C09136=1200.928,251.672,-63.247,-177.101,6.857,148.420
C09137=1200.933,251.424,-63.219,-177.103,6.855,148.421
C09138=1200.938,251.175,-63.192,-177.105,6.853,148.421
C09139=1200.942,250.926,-63.167,-177.109,6.850,148.421
C09140=1200.947,250.678,-63.140,-177.111,6.848,148.421
C09141=1200.951,250.429,-63.112,-177.113,6.846,148.421
C09142=1200.955,250.180,-63.086,-177.116,6.843,148.421
C09143=1200.959,249.932,-63.059,-177.119,6.841,148.422
C09144=1200.964,249.683,-63.033,-177.121,6.839,148.422
C09145=1200.968,249.435,-63.006,-177.124,6.836,148.422
C09146=1200.973,249.186,-62.979,-177.126,6.834,148.422
C09147=1200.977,248.938,-62.952,-177.129,6.832,148.422
C09148=1200.982,248.689,-62.926,-177.131,6.830,148.423
C09149=1200.986,248.441,-62.900,-177.134,6.828,148.423
C09150=1200.990,248.192,-62.872,-177.136,6.825,148.423
C09151=1200.995,247.943,-62.846,-177.139,6.824,148.423
C09152=1200.999,247.695,-62.820,-177.142,6.821,148.423
C09153=1201.004,247.446,-62.793,-177.144,6.819,148.424
C09154=1201.009,247.198,-62.767,-177.147,6.817,148.424
C09155=1201.013,246.950,-62.740,-177.150,6.814,148.424
C09156=1201.017,246.702,-62.714,-177.152,6.812,148.424
C09157=1201.022,246.452,-62.687,-177.154,6.810,148.424
C09158=1201.026,246.204,-62.661,-177.157,6.808,148.424
C09159=1201.031,245.955,-62.635,-177.160,6.805,148.425
C09160=1201.035,245.707,-62.608,-177.162,6.803,148.425
C09161=1201.040,245.458,-62.581,-177.165,6.801,148.425
C09162=1201.044,245.210,-62.555,-177.168,6.798,148.425
C09163=1201.049,244.961,-62.528,-177.170,6.796,148.426
C09164=1201.053,244.712,-62.502,-177.173,6.794,148.426
C09165=1201.057,244.464,-62.475,-177.175,6.792,148.426
C09166=1201.062,244.215,-62.450,-177.178,6.789,148.426
C09167=1201.066,243.967,-62.423,-177.180,6.787,148.426
C09168=1201.071,243.718,-62.397,-177.183,6.785,148.427
C09169=1201.075,243.470,-62.371,-177.186,6.783,148.427
C09170=1201.080,243.221,-62.344,-177.188,6.781,148.427
C09171=1201.084,242.973,-62.318,-177.191,6.779,148.427
C09172=1201.089,242.724,-62.292,-177.193,6.777,148.427
C09173=1201.093,242.475,-62.266,-177.196,6.774,148.428
C09174=1201.097,242.227,-62.239,-177.198,6.772,148.428
C09175=1201.102,241.978,-62.213,-177.201,6.770,148.428
C09176=1201.106,241.730,-62.187,-177.203,6.768,148.428
C09177=1201.111,241.480,-62.160,-177.206,6.765,148.428
C09178=1201.116,241.232,-62.135,-177.209,6.763,148.429
C09179=1201.120,240.984,-62.108,-177.211,6.761,148.429
C09180=1201.125,240.735,-62.082,-177.214,6.759,148.429
C09181=1201.129,240.486,-62.056,-177.217,6.757,148.429
C09182=1201.133,240.238,-62.030,-177.219,6.754,148.430
C09183=1201.138,239.989,-62.003,-177.222,6.752,148.430
C09184=1201.143,239.741,-61.978,-177.224,6.750,148.430
C09185=1201.146,239.493,-61.952,-177.227,6.748,148.430
C09186=1201.151,239.243,-61.925,-177.230,6.746,148.431
C09187=1201.156,238.995,-61.899,-177.232,6.744,148.431
C09188=1201.160,238.746,-61.874,-177.234,6.742,148.431
C09189=1201.164,238.498,-61.848,-177.237,6.739,148.431
C09190=1201.169,238.249,-61.821,-177.240,6.737,148.431
C09191=1201.174,238.000,-61.796,-177.242,6.735,148.432
C09192=1201.178,237.752,-61.770,-177.244,6.733,148.432
C09193=1201.182,237.503,-61.743,-177.248,6.730,148.432
C09194=1201.188,237.232,-61.715,-177.250,6.728,148.432
C09195=1201.192,236.960,-61.687,-177.253,6.725,148.432
C09196=1201.197,236.689,-61.658,-177.256,6.724,148.433
C09197=1201.202,236.418,-61.631,-177.259,6.721,148.433
C09198=1201.206,236.169,-61.605,-177.262,6.719,148.433
C09199=1201.211,235.920,-61.578,-177.264,6.717,148.434
C09200=1201.215,235.671,-61.552,-177.266,6.715,148.434
C09201=1201.220,235.423,-61.527,-177.269,6.712,148.434
C09202=1201.224,235.175,-61.501,-177.272,6.710,148.434
C09203=1201.228,234.926,-61.475,-177.274,6.708,148.435
C09204=1201.233,234.677,-61.449,-177.276,6.706,148.435
C09205=1201.238,234.429,-61.423,-177.280,6.704,148.435
C09206=1201.242,234.180,-61.398,-177.282,6.702,148.435
C09207=1201.247,233.931,-61.372,-177.284,6.700,148.435
C09208=1201.252,233.683,-61.346,-177.287,6.698,148.436
C09209=1201.256,233.434,-61.321,-177.290,6.696,148.436
C09210=1201.260,233.185,-61.295,-177.292,6.693,148.436
C09211=1201.264,232.936,-61.269,-177.295,6.691,148.436
C09212=1201.269,232.688,-61.244,-177.298,6.689,148.437
C09213=1201.273,232.440,-61.218,-177.300,6.687,148.437
C09214=1201.278,232.190,-61.192,-177.302,6.685,148.437
C09215=1201.283,231.942,-61.166,-177.306,6.683,148.437
C09216=1201.287,231.694,-61.141,-177.308,6.680,148.438
C09217=1201.292,231.445,-61.115,-177.310,6.679,148.438
C09218=1201.296,231.197,-61.089,-177.313,6.677,148.438
C09219=1201.301,230.947,-61.064,-177.315,6.675,148.438
C09220=1201.305,230.698,-61.039,-177.318,6.672,148.439
C09221=1201.310,230.450,-61.013,-177.321,6.670,148.439
C09222=1201.314,230.201,-60.988,-177.323,6.668,148.439
C09223=1201.318,229.953,-60.962,-177.326,6.666,148.439
C09224=1201.323,229.705,-60.936,-177.329,6.664,148.440
C09225=1201.327,229.456,-60.911,-177.331,6.662,148.440
C09226=1201.333,229.207,-60.886,-177.334,6.659,148.440
C09227=1201.337,228.958,-60.860,-177.337,6.658,148.440
C09228=1201.341,228.709,-60.834,-177.339,6.656,148.441
C09229=1201.346,228.461,-60.809,-177.341,6.654,148.441
C09230=1201.350,228.212,-60.784,-177.344,6.652,148.441
C09231=1201.355,227.963,-60.758,-177.347,6.649,148.441
C09232=1201.359,227.715,-60.733,-177.349,6.647,148.442
C09233=1201.364,227.466,-60.707,-177.352,6.645,148.442
C09234=1201.369,227.217,-60.683,-177.355,6.643,148.442
C09235=1201.372,226.969,-60.657,-177.357,6.641,148.442
C09236=1201.376,226.720,-60.632,-177.359,6.639,148.443
C09237=1201.381,226.472,-60.606,-177.363,6.637,148.443
C09238=1201.386,226.223,-60.581,-177.365,6.635,148.443
C09239=1201.391,225.975,-60.556,-177.367,6.633,148.443
C09240=1201.395,225.726,-60.530,-177.370,6.631,148.444
C09241=1201.400,225.477,-60.505,-177.373,6.629,148.444
C09242=1201.404,225.228,-60.480,-177.375,6.627,148.444
C09243=1201.409,224.979,-60.455,-177.378,6.624,148.444
C09244=1201.413,224.731,-60.430,-177.381,6.622,148.445
C09245=1201.417,224.482,-60.404,-177.383,6.620,148.445
C09246=1201.422,224.233,-60.379,-177.386,6.619,148.445
C09247=1201.426,223.985,-60.354,-177.388,6.616,148.445
C09248=1201.432,223.736,-60.329,-177.391,6.615,148.446
C09249=1201.436,223.487,-60.303,-177.394,6.612,148.446
C09250=1201.440,223.239,-60.279,-177.396,6.610,148.446
C09251=1201.444,222.990,-60.253,-177.399,6.608,148.447
C09252=1201.450,222.741,-60.229,-177.401,6.606,148.447
C09253=1201.454,222.492,-60.203,-177.404,6.604,148.447
C09254=1201.459,222.244,-60.178,-177.407,6.602,148.448
C09255=1201.462,221.995,-60.153,-177.409,6.600,148.448
C09256=1201.468,221.746,-60.128,-177.412,6.598,148.448
C09257=1201.472,221.498,-60.103,-177.415,6.596,148.448
C09258=1201.477,221.249,-60.078,-177.417,6.594,148.449
C09259=1201.480,221.000,-60.053,-177.420,6.592,148.449
C09260=1201.485,220.752,-60.028,-177.422,6.590,148.449
C09261=1201.490,220.503,-60.002,-177.425,6.588,148.449
C09262=1201.494,220.254,-59.978,-177.427,6.586,148.450
C09263=1201.499,220.006,-59.954,-177.430,6.583,148.450
C09264=1201.503,219.757,-59.928,-177.433,6.581,148.450
C09265=1201.509,219.508,-59.903,-177.435,6.580,148.450
C09266=1201.512,219.259,-59.879,-177.438,6.578,148.451
C09267=1201.517,219.011,-59.853,-177.441,6.576,148.451
C09268=1201.522,218.762,-59.828,-177.443,6.574,148.451
C09269=1201.526,218.513,-59.804,-177.446,6.572,148.452
C09270=1201.530,218.264,-59.779,-177.448,6.570,148.452
C09271=1201.535,218.016,-59.754,-177.451,6.567,148.452
C09272=1201.540,217.767,-59.730,-177.454,6.565,148.452
C09273=1201.544,217.518,-59.704,-177.456,6.563,148.453
C09274=1201.549,217.270,-59.680,-177.459,6.562,148.453
C09275=1201.553,217.021,-59.655,-177.461,6.560,148.453
C09276=1201.558,216.772,-59.630,-177.464,6.558,148.454
C09277=1201.562,216.524,-59.606,-177.467,6.556,148.454
C09278=1201.567,216.275,-59.581,-177.469,6.554,148.454
C09279=1201.571,216.026,-59.556,-177.472,6.551,148.454
C09280=1201.576,215.777,-59.531,-177.475,6.550,148.455
C09281=1201.581,215.528,-59.507,-177.477,6.548,148.455
C09282=1201.585,215.280,-59.482,-177.480,6.546,148.455
C09283=1201.589,215.031,-59.457,-177.482,6.544,148.455
C09284=1201.594,214.782,-59.433,-177.485,6.542,148.456
C09285=1201.599,214.534,-59.408,-177.488,6.540,148.456
C09286=1201.603,214.285,-59.384,-177.490,6.538,148.456
C09287=1201.608,214.036,-59.359,-177.493,6.536,148.457
C09288=1201.612,213.787,-59.335,-177.496,6.534,148.457
C09289=1201.617,213.538,-59.310,-177.498,6.532,148.457
C09290=1201.621,213.290,-59.285,-177.501,6.530,148.458
C09291=1201.626,213.042,-59.261,-177.503,6.528,148.458
C09292=1201.630,212.792,-59.236,-177.506,6.526,148.458
C09293=1201.635,212.544,-59.211,-177.509,6.524,148.459
C09294=1201.639,212.295,-59.187,-177.511,6.522,148.459
C09295=1201.644,212.046,-59.162,-177.514,6.520,148.459
C09296=1201.648,211.797,-59.138,-177.516,6.518,148.459
C09297=1201.653,211.549,-59.114,-177.519,6.517,148.460
C09298=1201.658,211.278,-59.086,-177.522,6.514,148.460
C09299=1201.663,211.007,-59.061,-177.525,6.512,148.460
C09300=1201.668,210.737,-59.034,-177.527,6.510,148.461
C09301=1201.673,210.467,-59.008,-177.531,6.508,148.461
C09302=1201.678,210.218,-58.983,-177.533,6.506,148.461
C09303=1201.682,209.969,-58.959,-177.536,6.504,148.462
C09304=1201.686,209.721,-58.934,-177.539,6.502,148.462
C09305=1201.691,209.472,-58.910,-177.541,6.500,148.462
C09306=1201.695,209.223,-58.885,-177.543,6.498,148.462
C09307=1201.700,208.974,-58.862,-177.546,6.496,148.463
C09308=1201.705,208.725,-58.837,-177.549,6.495,148.463
C09309=1201.709,208.477,-58.813,-177.551,6.493,148.463
C09310=1201.715,208.228,-58.789,-177.554,6.491,148.464
C09311=1201.718,207.979,-58.764,-177.557,6.488,148.464
C09312=1201.723,207.731,-58.740,-177.560,6.486,148.464
C09313=1201.728,207.482,-58.715,-177.562,6.484,148.465
C09314=1201.733,207.233,-58.692,-177.565,6.482,148.465
C09315=1201.736,206.984,-58.668,-177.567,6.481,148.465
C09316=1201.742,206.735,-58.643,-177.570,6.479,148.466
C09317=1201.746,206.487,-58.619,-177.573,6.477,148.466
C09318=1201.751,206.237,-58.595,-177.575,6.475,148.466
C09319=1201.755,205.989,-58.571,-177.578,6.473,148.467
C09320=1201.760,205.740,-58.546,-177.581,6.472,148.467
C09321=1201.764,205.491,-58.522,-177.583,6.469,148.467
C09322=1201.769,205.242,-58.499,-177.585,6.468,148.467
C09323=1201.774,204.993,-58.474,-177.588,6.466,148.468
C09324=1201.778,204.745,-58.450,-177.591,6.464,148.468
C09325=1201.783,204.496,-58.427,-177.593,6.462,148.468
C09326=1201.787,204.247,-58.402,-177.596,6.460,148.469
C09327=1201.791,203.999,-58.378,-177.599,6.458,148.469
C09328=1201.797,203.749,-58.354,-177.601,6.457,148.469
C09329=1201.801,203.501,-58.330,-177.604,6.455,148.470
C09330=1201.805,203.252,-58.306,-177.606,6.453,148.470
C09331=1201.810,203.003,-58.283,-177.609,6.451,148.470
C09332=1201.814,202.755,-58.259,-177.611,6.449,148.471
C09333=1201.819,202.505,-58.234,-177.615,6.446,148.471
C09334=1201.824,202.256,-58.210,-177.617,6.445,148.471
C09335=1201.828,202.008,-58.186,-177.620,6.443,148.472
C09336=1201.833,201.759,-58.163,-177.623,6.441,148.472
C09337=1201.837,201.511,-58.139,-177.625,6.439,148.472
C09338=1201.842,201.262,-58.116,-177.628,6.437,148.473
C09339=1201.847,201.013,-58.091,-177.630,6.435,148.473
C09340=1201.852,200.764,-58.068,-177.633,6.434,148.473
C09341=1201.855,200.515,-58.043,-177.635,6.431,148.473
C09342=1201.860,200.266,-58.020,-177.638,6.430,148.474
C09343=1201.865,200.017,-57.996,-177.641,6.428,148.474
C09344=1201.869,199.768,-57.972,-177.643,6.426,148.474
C09345=1201.874,199.520,-57.948,-177.646,6.424,148.475
C09346=1201.878,199.271,-57.925,-177.649,6.422,148.475
C09347=1201.883,199.022,-57.901,-177.651,6.421,148.475
C09348=1201.887,198.773,-57.877,-177.654,6.419,148.476
C09349=1201.892,198.525,-57.853,-177.657,6.417,148.476
C09350=1201.897,198.276,-57.829,-177.659,6.415,148.477
C09351=1201.902,198.027,-57.806,-177.662,6.413,148.477
C09352=1201.906,197.778,-57.782,-177.664,6.411,148.477
C09353=1201.911,197.529,-57.759,-177.667,6.410,148.478
C09354=1201.915,197.281,-57.735,-177.670,6.408,148.478
C09355=1201.920,197.032,-57.711,-177.672,6.406,148.478
C09356=1201.925,196.783,-57.688,-177.675,6.404,148.478
C09357=1201.929,196.534,-57.664,-177.677,6.402,148.479
C09358=1201.934,196.285,-57.640,-177.680,6.400,148.479
C09359=1201.939,196.036,-57.617,-177.683,6.398,148.479
C09360=1201.943,195.787,-57.594,-177.685,6.397,148.480
C09361=1201.948,195.539,-57.570,-177.688,6.395,148.480
C09362=1201.952,195.290,-57.546,-177.691,6.393,148.480
C09363=1201.957,195.041,-57.523,-177.693,6.391,148.481
C09364=1201.962,194.792,-57.499,-177.696,6.389,148.481
C09365=1201.966,194.543,-57.475,-177.698,6.388,148.482
C09366=1201.970,194.294,-57.453,-177.701,6.387,148.482
C09367=1201.975,194.045,-57.429,-177.703,6.385,148.482
C09368=1201.980,193.796,-57.406,-177.706,6.383,148.483
C09369=1201.984,193.548,-57.382,-177.709,6.381,148.483
C09370=1201.989,193.299,-57.358,-177.711,6.379,148.483
C09371=1201.993,193.050,-57.335,-177.714,6.377,148.484
C09372=1201.998,192.801,-57.312,-177.717,6.376,148.484
C09373=1202.003,192.552,-57.288,-177.719,6.374,148.484
C09374=1202.007,192.303,-57.265,-177.722,6.372,148.485
C09375=1202.012,192.054,-57.241,-177.724,6.370,148.485
C09376=1202.016,191.806,-57.218,-177.727,6.368,148.485
C09377=1202.021,191.557,-57.195,-177.730,6.367,148.486
C09378=1202.025,191.308,-57.172,-177.732,6.365,148.486
C09379=1202.030,191.059,-57.148,-177.735,6.363,148.486
C09380=1202.035,190.810,-57.125,-177.738,6.361,148.487
C09381=1202.040,190.561,-57.102,-177.740,6.359,148.487
C09382=1202.045,190.312,-57.078,-177.743,6.357,148.487
C09383=1202.049,190.063,-57.056,-177.746,6.356,148.488
C09384=1202.053,189.814,-57.032,-177.748,6.354,148.488
C09385=1202.058,189.565,-57.009,-177.751,6.352,148.489
C09386=1202.063,189.316,-56.986,-177.754,6.350,148.489
C09387=1202.067,189.067,-56.962,-177.756,6.349,148.489
C09388=1202.071,188.819,-56.939,-177.758,6.347,148.490
C09389=1202.077,188.570,-56.916,-177.761,6.346,148.490
C09390=1202.081,188.321,-56.893,-177.764,6.344,148.490
C09391=1202.086,188.072,-56.870,-177.766,6.342,148.491
C09392=1202.090,187.823,-56.847,-177.769,6.340,148.491
C09393=1202.095,187.574,-56.824,-177.772,6.338,148.491
C09394=1202.099,187.325,-56.800,-177.774,6.337,148.492
C09395=1202.104,187.076,-56.777,-177.777,6.335,148.492
C09396=1202.109,186.828,-56.755,-177.780,6.333,148.492
C09397=1202.113,186.579,-56.731,-177.782,6.331,148.493
C09398=1202.118,186.330,-56.708,-177.785,6.329,148.493
C09399=1202.122,186.082,-56.685,-177.788,6.328,148.493
C09400=1202.127,185.832,-56.662,-177.790,6.326,148.494
C09401=1202.132,185.583,-56.639,-177.792,6.325,148.494
C09402=1202.136,185.313,-56.615,-177.796,6.322,148.495
C09403=1202.142,185.044,-56.590,-177.798,6.320,148.495
C09404=1202.147,184.775,-56.564,-177.801,6.318,148.495
C09405=1202.151,184.505,-56.539,-177.804,6.317,148.496
C09406=1202.157,184.256,-56.517,-177.806,6.315,148.496
C09407=1202.161,184.007,-56.494,-177.809,6.313,148.496
C09408=1202.166,183.758,-56.471,-177.812,6.312,148.497
C09409=1202.170,183.509,-56.448,-177.815,6.310,148.497
C09410=1202.174,183.260,-56.426,-177.817,6.308,148.498
C09411=1202.180,183.012,-56.403,-177.820,6.307,148.498
C09412=1202.184,182.763,-56.379,-177.822,6.305,148.498
C09413=1202.188,182.514,-56.356,-177.825,6.303,148.499
C09414=1202.193,182.264,-56.334,-177.828,6.302,148.499
C09415=1202.198,182.016,-56.311,-177.830,6.300,148.499
C09416=1202.203,181.767,-56.288,-177.833,6.298,148.500
C09417=1202.207,181.518,-56.266,-177.836,6.296,148.500
C09418=1202.212,181.269,-56.243,-177.838,6.294,148.500
C09419=1202.216,181.021,-56.220,-177.841,6.292,148.501
C09420=1202.221,180.771,-56.198,-177.843,6.292,148.501
C09421=1202.226,180.522,-56.174,-177.846,6.290,148.502
C09422=1202.230,180.273,-56.151,-177.848,6.288,148.502
C09423=1202.236,180.024,-56.129,-177.851,6.286,148.502
C09424=1202.239,179.776,-56.106,-177.854,6.284,148.503
C09425=1202.244,179.526,-56.084,-177.856,6.282,148.503
C09426=1202.249,179.278,-56.061,-177.859,6.281,148.503
C09427=1202.254,179.029,-56.038,-177.862,6.279,148.504
C09428=1202.258,178.780,-56.016,-177.864,6.278,148.504
C09429=1202.263,178.531,-55.993,-177.867,6.276,148.505
C09430=1202.268,178.282,-55.971,-177.869,6.275,148.505
C09431=1202.272,178.033,-55.948,-177.872,6.273,148.505
C09432=1202.277,177.784,-55.926,-177.875,6.271,148.506
C09433=1202.281,177.536,-55.903,-177.877,6.269,148.506
C09434=1202.286,177.286,-55.881,-177.880,6.267,148.506
C09435=1202.290,177.037,-55.858,-177.882,6.266,148.507
C09436=1202.296,176.788,-55.835,-177.885,6.265,148.507
C09437=1202.300,176.540,-55.813,-177.888,6.263,148.508
C09438=1202.305,176.291,-55.791,-177.890,6.261,148.508
C09439=1202.309,176.042,-55.768,-177.893,6.259,148.508
C09440=1202.313,175.793,-55.746,-177.896,6.257,148.509
C09441=1202.319,175.544,-55.723,-177.898,6.256,148.509
C09442=1202.323,175.295,-55.701,-177.901,6.255,148.510
C09443=1202.327,175.046,-55.679,-177.903,6.253,148.510
C09444=1202.333,174.797,-55.656,-177.906,6.251,148.510
C09445=1202.337,174.548,-55.633,-177.909,6.250,148.511
C09446=1202.343,174.299,-55.611,-177.911,6.248,148.511
C09447=1202.346,174.050,-55.588,-177.914,6.246,148.511
C09448=1202.351,173.801,-55.566,-177.916,6.245,148.512
C09449=1202.356,173.552,-55.544,-177.919,6.243,148.512
C09450=1202.360,173.303,-55.521,-177.922,6.241,148.513
C09451=1202.365,173.055,-55.500,-177.924,6.240,148.513
C09452=1202.369,172.805,-55.478,-177.927,6.238,148.513
C09453=1202.374,172.556,-55.454,-177.930,6.236,148.514
C09454=1202.379,172.308,-55.433,-177.932,6.235,148.514
C09455=1202.383,172.058,-55.411,-177.935,6.233,148.515
C09456=1202.389,171.809,-55.388,-177.937,6.232,148.515
C09457=1202.393,171.561,-55.365,-177.940,6.230,148.515
C09458=1202.398,171.312,-55.344,-177.943,6.228,148.516
C09459=1202.402,171.063,-55.322,-177.945,6.227,148.516
C09460=1202.407,170.813,-55.299,-177.948,6.225,148.516
C09461=1202.412,170.564,-55.277,-177.951,6.224,148.517
C09462=1202.416,170.316,-55.255,-177.953,6.222,148.517
C09463=1202.421,170.067,-55.233,-177.956,6.220,148.518
C09464=1202.426,169.817,-55.210,-177.959,6.218,148.518
C09465=1202.431,169.569,-55.189,-177.961,6.217,148.518
C09466=1202.435,169.319,-55.167,-177.963,6.216,148.519
C09467=1202.440,169.071,-55.145,-177.966,6.214,148.519
C09468=1202.444,168.822,-55.122,-177.969,6.212,148.520
C09469=1202.449,168.573,-55.100,-177.972,6.211,148.520
C09470=1202.454,168.324,-55.078,-177.974,6.210,148.521
C09471=1202.458,168.075,-55.056,-177.977,6.208,148.521
C09472=1202.463,167.826,-55.034,-177.979,6.206,148.521
C09473=1202.468,167.577,-55.012,-177.982,6.204,148.522
C09474=1202.473,167.327,-54.990,-177.984,6.203,148.522
C09475=1202.477,167.079,-54.968,-177.987,6.201,148.522
C09476=1202.482,166.829,-54.946,-177.990,6.200,148.523
C09477=1202.487,166.581,-54.924,-177.993,6.198,148.523
C09478=1202.491,166.331,-54.902,-177.995,6.196,148.524
C09479=1202.496,166.083,-54.881,-177.997,6.195,148.524
C09480=1202.500,165.833,-54.859,-178.000,6.194,148.524
C09481=1202.505,165.585,-54.837,-178.003,6.192,148.525
C09482=1202.510,165.336,-54.815,-178.005,6.190,148.525
C09483=1202.515,165.086,-54.793,-178.009,6.189,148.526
C09484=1202.520,164.838,-54.771,-178.011,6.188,148.526
C09485=1202.524,164.588,-54.749,-178.013,6.186,148.527
C09486=1202.529,164.340,-54.727,-178.016,6.184,148.527
C09487=1202.533,164.091,-54.705,-178.019,6.182,148.527
C09488=1202.538,163.842,-54.683,-178.021,6.181,148.528
C09489=1202.542,163.593,-54.661,-178.024,6.180,148.528
C09490=1202.547,163.344,-54.640,-178.027,6.178,148.529
C09491=1202.552,163.095,-54.618,-178.029,6.176,148.529
C09492=1202.556,162.846,-54.596,-178.031,6.175,148.529
C09493=1202.561,162.597,-54.575,-178.034,6.173,148.530
C09494=1202.566,162.347,-54.553,-178.037,6.172,148.530
C09495=1202.570,162.099,-54.531,-178.040,6.170,148.531
C09496=1202.575,161.850,-54.510,-178.042,6.169,148.531
C09497=1202.580,161.601,-54.488,-178.045,6.167,148.531
C09498=1202.584,161.352,-54.466,-178.047,6.166,148.532
C09499=1202.589,161.102,-54.445,-178.050,6.164,148.532
C09500=1202.594,160.853,-54.423,-178.052,6.163,148.533
C09501=1202.599,160.605,-54.401,-178.055,6.161,148.533
C09502=1202.603,160.355,-54.379,-178.058,6.160,148.534
C09503=1202.608,160.107,-54.357,-178.061,6.158,148.534
C09504=1202.613,159.858,-54.336,-178.063,6.157,148.534
C09505=1202.617,159.608,-54.314,-178.065,6.155,148.535
C09506=1202.622,159.339,-54.292,-178.069,6.154,148.535
C09507=1202.627,159.070,-54.268,-178.071,6.152,148.536
C09508=1202.632,158.801,-54.245,-178.074,6.150,148.536
C09509=1202.637,158.532,-54.221,-178.077,6.149,148.537
C09510=1202.642,158.283,-54.200,-178.080,6.147,148.537
C09511=1202.647,158.035,-54.178,-178.082,6.146,148.537
C09512=1202.652,157.785,-54.157,-178.085,6.144,148.538
C09513=1202.656,157.536,-54.136,-178.088,6.143,148.538
C09514=1202.661,157.288,-54.114,-178.090,6.141,148.539
C09515=1202.666,157.039,-54.093,-178.092,6.140,148.539
C09516=1202.670,156.789,-54.071,-178.095,6.138,148.540
C09517=1202.675,156.540,-54.050,-178.098,6.137,148.540
C09518=1202.680,156.291,-54.028,-178.101,6.135,148.540
C09519=1202.685,156.042,-54.006,-178.103,6.134,148.541
C09520=1202.689,155.793,-53.986,-178.106,6.132,148.541
C09521=1202.694,155.544,-53.964,-178.108,6.130,148.542
C09522=1202.699,155.295,-53.943,-178.111,6.130,148.542
C09523=1202.703,155.046,-53.921,-178.114,6.128,148.543
C09524=1202.708,154.797,-53.900,-178.116,6.126,148.543
C09525=1202.713,154.548,-53.879,-178.119,6.124,148.543
C09526=1202.717,154.300,-53.857,-178.121,6.123,148.544
C09527=1202.722,154.050,-53.836,-178.124,6.122,148.544
C09528=1202.727,153.801,-53.814,-178.127,6.120,148.545
C09529=1202.732,153.552,-53.793,-178.129,6.119,148.545
C09530=1202.736,153.303,-53.772,-178.132,6.117,148.546
C09531=1202.741,153.053,-53.751,-178.135,6.116,148.546
C09532=1202.746,152.804,-53.730,-178.137,6.115,148.547
C09533=1202.751,152.555,-53.708,-178.140,6.113,148.547
C09534=1202.755,152.307,-53.688,-178.142,6.111,148.547
C09535=1202.760,152.058,-53.666,-178.146,6.110,148.548
C09536=1202.765,151.808,-53.645,-178.148,6.109,148.548
C09537=1202.769,151.560,-53.624,-178.150,6.107,148.549
C09538=1202.774,151.310,-53.603,-178.153,6.105,148.549
C09539=1202.779,151.061,-53.582,-178.156,6.105,148.550
C09540=1202.784,150.812,-53.560,-178.158,6.103,148.550
C09541=1202.788,150.563,-53.540,-178.161,6.101,148.550
C09542=1202.793,150.314,-53.518,-178.163,6.100,148.551
C09543=1202.798,150.065,-53.497,-178.166,6.099,148.551
C09544=1202.802,149.816,-53.477,-178.169,6.097,148.552
C09545=1202.807,149.567,-53.455,-178.171,6.096,148.552
C09546=1202.812,149.317,-53.434,-178.174,6.094,148.553
C09547=1202.816,149.068,-53.413,-178.177,6.093,148.553
C09548=1202.821,148.819,-53.392,-178.179,6.092,148.554
C09549=1202.826,148.571,-53.371,-178.182,6.090,148.554
C09550=1202.831,148.322,-53.350,-178.184,6.088,148.554
C09551=1202.836,148.072,-53.329,-178.187,6.088,148.555
C09552=1202.840,147.824,-53.308,-178.190,6.086,148.555
C09553=1202.845,147.574,-53.287,-178.192,6.084,148.556
C09554=1202.849,147.325,-53.266,-178.194,6.083,148.556
C09555=1202.854,147.076,-53.245,-178.198,6.082,148.557
C09556=1202.859,146.827,-53.224,-178.200,6.080,148.557
C09557=1202.864,146.578,-53.203,-178.202,6.079,148.557
C09558=1202.869,146.329,-53.182,-178.205,6.077,148.558
C09559=1202.873,146.080,-53.162,-178.208,6.076,148.558
C09560=1202.878,145.831,-53.141,-178.210,6.075,148.559
C09561=1202.883,145.582,-53.121,-178.213,6.073,148.559
C09562=1202.887,145.332,-53.099,-178.216,6.071,148.560
C09563=1202.891,145.084,-53.078,-178.218,6.070,148.560
C09564=1202.897,144.834,-53.057,-178.221,6.069,148.561
C09565=1202.901,144.585,-53.037,-178.223,6.068,148.561
C09566=1202.906,144.336,-53.016,-178.226,6.066,148.562
C09567=1202.911,144.087,-52.996,-178.229,6.064,148.562
C09568=1202.916,143.838,-52.975,-178.231,6.063,148.562
C09569=1202.920,143.589,-52.954,-178.234,6.062,148.563
C09570=1202.925,143.340,-52.933,-178.237,6.060,148.563
C09571=1202.930,143.091,-52.913,-178.239,6.059,148.564
C09572=1202.935,142.842,-52.891,-178.242,6.058,148.564
C09573=1202.939,142.593,-52.871,-178.245,6.056,148.565
C09574=1202.944,142.344,-52.850,-178.247,6.055,148.565
C09575=1202.949,142.095,-52.830,-178.250,6.053,148.566
C09576=1202.953,141.845,-52.808,-178.252,6.053,148.566
C09577=1202.958,141.596,-52.788,-178.255,6.051,148.567
C09578=1202.962,141.347,-52.767,-178.258,6.049,148.567
C09579=1202.967,141.098,-52.746,-178.260,6.049,148.568
C09580=1202.972,140.849,-52.726,-178.263,6.047,148.568
C09581=1202.977,140.600,-52.705,-178.266,6.045,148.568
C09582=1202.982,140.351,-52.685,-178.268,6.044,148.569
C09583=1202.986,140.101,-52.665,-178.271,6.043,148.569
C09584=1202.991,139.852,-52.644,-178.273,6.042,148.570
C09585=1202.996,139.603,-52.624,-178.276,6.040,148.570
C09586=1203.001,139.354,-52.603,-178.279,6.038,148.571
C09587=1203.005,139.105,-52.582,-178.281,6.037,148.571
C09588=1203.010,138.856,-52.562,-178.284,6.036,148.571
C09589=1203.015,138.606,-52.541,-178.286,6.035,148.572
C09590=1203.020,138.357,-52.521,-178.289,6.033,148.573
C09591=1203.024,138.109,-52.500,-178.292,6.032,148.573
C09592=1203.030,137.860,-52.480,-178.294,6.031,148.574
C09593=1203.034,137.610,-52.460,-178.297,6.029,148.574
C09594=1203.039,137.361,-52.440,-178.299,6.028,148.574
C09595=1203.044,137.112,-52.419,-178.302,6.027,148.575
C09596=1203.049,136.863,-52.398,-178.305,6.025,148.575
C09597=1203.053,136.614,-52.378,-178.307,6.024,148.576
C09598=1203.058,136.364,-52.358,-178.310,6.023,148.576
C09599=1203.063,136.115,-52.337,-178.312,6.022,148.577
C09600=1203.067,135.866,-52.317,-178.315,6.020,148.577
C09601=1203.072,135.618,-52.297,-178.318,6.018,148.578
C09602=1203.077,135.368,-52.276,-178.320,6.017,148.578
C09603=1203.082,135.119,-52.256,-178.323,6.016,148.578
C09604=1203.086,134.870,-52.236,-178.325,6.015,148.579
C09605=1203.091,134.621,-52.215,-178.328,6.013,148.580
C09606=1203.096,134.371,-52.195,-178.330,6.012,148.580
C09607=1203.101,134.123,-52.175,-178.333,6.011,148.581
C09608=1203.106,133.874,-52.155,-178.336,6.009,148.581
C09609=1203.110,133.624,-52.135,-178.338,6.008,148.581
C09610=1203.116,133.356,-52.113,-178.341,6.007,148.582
C09611=1203.121,133.087,-52.092,-178.344,6.005,148.582
C09612=1203.125,132.818,-52.069,-178.347,6.004,148.583
C09613=1203.131,132.549,-52.047,-178.350,6.003,148.584
C09614=1203.136,132.301,-52.027,-178.353,6.001,148.584
C09615=1203.141,132.051,-52.007,-178.355,6.000,148.584
C09616=1203.145,131.802,-51.987,-178.358,5.999,148.585
C09617=1203.150,131.553,-51.967,-178.360,5.998,148.585
C09618=1203.154,131.304,-51.947,-178.363,5.996,148.586
C09619=1203.159,131.055,-51.927,-178.366,5.995,148.586
C09620=1203.164,130.805,-51.906,-178.368,5.994,148.587
C09621=1203.169,130.557,-51.886,-178.371,5.992,148.587
C09622=1203.174,130.308,-51.866,-178.373,5.991,148.588
C09623=1203.178,130.058,-51.846,-178.376,5.989,148.588
C09624=1203.183,129.809,-51.826,-178.379,5.989,148.589
C09625=1203.188,129.560,-51.806,-178.381,5.987,148.589
C09626=1203.192,129.311,-51.786,-178.383,5.986,148.590
C09627=1203.197,129.062,-51.767,-178.387,5.985,148.590
C09628=1203.202,128.813,-51.746,-178.389,5.983,148.591
C09629=1203.207,128.563,-51.726,-178.391,5.982,148.591
C09630=1203.212,128.314,-51.706,-178.394,5.981,148.592
C09631=1203.217,128.065,-51.686,-178.397,5.980,148.592
C09632=1203.222,127.816,-51.667,-178.400,5.978,148.593
C09633=1203.226,127.567,-51.646,-178.402,5.977,148.593
C09634=1203.231,127.317,-51.627,-178.405,5.975,148.593
C09635=1203.235,127.068,-51.606,-178.407,5.975,148.594
C09636=1203.241,126.819,-51.587,-178.410,5.973,148.594
C09637=1203.245,126.570,-51.567,-178.412,5.973,148.595
C09638=1203.250,126.321,-51.547,-178.415,5.971,148.596
C09639=1203.255,126.071,-51.527,-178.417,5.970,148.596
C09640=1203.259,125.822,-51.507,-178.420,5.968,148.597
C09641=1203.265,125.574,-51.488,-178.423,5.967,148.597
C09642=1203.269,125.324,-51.468,-178.425,5.966,148.597
C09643=1203.274,125.075,-51.448,-178.428,5.965,148.598
C09644=1203.278,124.825,-51.428,-178.431,5.963,148.598
C09645=1203.284,124.577,-51.409,-178.434,5.962,148.599
C09646=1203.288,124.328,-51.388,-178.436,5.961,148.599
C09647=1203.293,124.078,-51.369,-178.439,5.959,148.600
C09648=1203.298,123.829,-51.349,-178.441,5.959,148.600
C09649=1203.303,123.580,-51.329,-178.444,5.957,148.601
C09650=1203.307,123.331,-51.310,-178.446,5.956,148.601
C09651=1203.312,123.081,-51.290,-178.449,5.954,148.602
C09652=1203.317,122.833,-51.271,-178.452,5.954,148.602
C09653=1203.321,122.584,-51.251,-178.454,5.952,148.603
C09654=1203.326,122.334,-51.231,-178.457,5.951,148.603
C09655=1203.331,122.085,-51.212,-178.460,5.950,148.604
C09656=1203.336,121.836,-51.192,-178.462,5.949,148.604
C09657=1203.341,121.587,-51.172,-178.465,5.947,148.605
C09658=1203.346,121.338,-51.152,-178.467,5.946,148.605
C09659=1203.351,121.088,-51.133,-178.470,5.945,148.606
C09660=1203.355,120.839,-51.114,-178.472,5.944,148.606
C09661=1203.360,120.590,-51.094,-178.475,5.942,148.607
C09662=1203.365,120.341,-51.075,-178.478,5.942,148.607
C09663=1203.369,120.092,-51.054,-178.480,5.940,148.608
C09664=1203.375,119.843,-51.035,-178.483,5.939,148.608
C09665=1203.379,119.593,-51.015,-178.486,5.937,148.609
C09666=1203.383,119.344,-50.996,-178.488,5.937,148.609
C09667=1203.389,119.095,-50.977,-178.491,5.936,148.610
C09668=1203.393,118.845,-50.957,-178.493,5.934,148.610
C09669=1203.398,118.596,-50.938,-178.496,5.934,148.611
C09670=1203.403,118.347,-50.918,-178.499,5.932,148.611
C09671=1203.408,118.097,-50.899,-178.501,5.931,148.612
C09672=1203.412,117.850,-50.879,-178.504,5.929,148.612
C09673=1203.417,117.600,-50.860,-178.506,5.929,148.613
C09674=1203.422,117.350,-50.840,-178.509,5.927,148.613
C09675=1203.427,117.101,-50.821,-178.511,5.926,148.614
C09676=1203.431,116.852,-50.802,-178.514,5.925,148.614
C09677=1203.437,116.603,-50.782,-178.517,5.924,148.615
C09678=1203.441,116.354,-50.763,-178.520,5.922,148.615
C09679=1203.446,116.104,-50.743,-178.522,5.921,148.616
C09680=1203.451,115.856,-50.724,-178.525,5.920,148.616
C09681=1203.455,115.606,-50.705,-178.527,5.919,148.617
C09682=1203.461,115.357,-50.685,-178.530,5.918,148.618
C09683=1203.466,115.108,-50.666,-178.532,5.917,148.618
C09684=1203.470,114.858,-50.647,-178.535,5.916,148.618
C09685=1203.475,114.609,-50.628,-178.538,5.914,148.619
C09686=1203.480,114.359,-50.609,-178.540,5.913,148.619
C09687=1203.485,114.111,-50.590,-178.543,5.912,148.620
C09688=1203.489,113.861,-50.570,-178.545,5.911,148.620
C09689=1203.495,113.612,-50.551,-178.548,5.910,148.621
C09690=1203.499,113.363,-50.532,-178.550,5.909,148.621
C09691=1203.504,113.114,-50.513,-178.554,5.907,148.622
C09692=1203.509,112.865,-50.493,-178.556,5.906,148.623
C09693=1203.513,112.616,-50.474,-178.558,5.906,148.623
C09694=1203.518,112.366,-50.455,-178.561,5.904,148.624
C09695=1203.524,112.117,-50.436,-178.564,5.903,148.624
C09696=1203.528,111.868,-50.417,-178.566,5.902,148.625
C09697=1203.533,111.619,-50.398,-178.569,5.901,148.625
C09698=1203.538,111.369,-50.378,-178.572,5.899,148.626
C09699=1203.542,111.119,-50.360,-178.574,5.898,148.626
C09700=1203.548,110.871,-50.340,-178.577,5.897,148.627
C09701=1203.552,110.621,-50.321,-178.579,5.896,148.627
C09702=1203.557,110.373,-50.302,-178.582,5.895,148.628
C09703=1203.562,110.124,-50.283,-178.584,5.894,148.628
C09704=1203.567,109.874,-50.264,-178.587,5.893,148.629
C09705=1203.572,109.625,-50.245,-178.590,5.891,148.629
C09706=1203.576,109.376,-50.226,-178.592,5.891,148.630
C09707=1203.582,109.126,-50.207,-178.595,5.890,148.630
C09708=1203.586,108.877,-50.188,-178.598,5.888,148.631
C09709=1203.591,108.628,-50.169,-178.600,5.887,148.631
C09710=1203.595,108.379,-50.150,-178.603,5.886,148.632
C09711=1203.601,108.129,-50.131,-178.605,5.885,148.632
C09712=1203.605,107.880,-50.112,-178.608,5.884,148.633
C09713=1203.610,107.631,-50.093,-178.610,5.883,148.633
C09714=1203.615,107.362,-50.073,-178.614,5.881,148.634
C09715=1203.620,107.094,-50.053,-178.616,5.881,148.635
C09716=1203.626,106.826,-50.033,-178.619,5.879,148.635
C09717=1203.631,106.557,-50.011,-178.622,5.878,148.636
C09718=1203.636,106.308,-49.993,-178.625,5.877,148.636
C09719=1203.640,106.058,-49.974,-178.627,5.876,148.637
C09720=1203.645,105.810,-49.955,-178.630,5.875,148.637
C09721=1203.651,105.560,-49.937,-178.632,5.874,148.638
C09722=1203.655,105.311,-49.917,-178.635,5.873,148.638
C09723=1203.659,105.062,-49.900,-178.638,5.871,148.639
C09724=1203.664,104.812,-49.880,-178.640,5.871,148.639
C09725=1203.669,104.563,-49.862,-178.643,5.869,148.640
C09726=1203.674,104.314,-49.843,-178.645,5.868,148.641
C09727=1203.679,104.064,-49.824,-178.648,5.867,148.641
C09728=1203.684,103.815,-49.805,-178.651,5.866,148.642
C09729=1203.688,103.566,-49.787,-178.653,5.865,148.642
C09730=1203.693,103.317,-49.768,-178.656,5.865,148.643
C09731=1203.699,103.068,-49.749,-178.658,5.863,148.643
C09732=1203.703,102.818,-49.730,-178.661,5.862,148.644
C09733=1203.708,102.569,-49.712,-178.664,5.860,148.644
C09734=1203.713,102.320,-49.693,-178.666,5.860,148.645
C09735=1203.717,102.070,-49.675,-178.668,5.859,148.645
C09736=1203.723,101.822,-49.655,-178.671,5.858,148.646
C09737=1203.727,101.572,-49.637,-178.674,5.857,148.646
C09738=1203.731,101.323,-49.618,-178.676,5.856,148.647
C09739=1203.737,101.074,-49.600,-178.679,5.854,148.647
C09740=1203.742,100.824,-49.582,-178.682,5.854,148.648
C09741=1203.746,100.575,-49.563,-178.684,5.852,148.648
C09742=1203.752,100.326,-49.544,-178.687,5.851,148.649
C09743=1203.756,100.077,-49.525,-178.689,5.850,148.649
C09744=1203.761,99.827,-49.507,-178.692,5.849,148.650
C09745=1203.766,99.578,-49.489,-178.695,5.848,148.651
C09746=1203.771,99.329,-49.470,-178.697,5.847,148.651
C09747=1203.775,99.079,-49.451,-178.700,5.846,148.652
C09748=1203.781,98.830,-49.433,-178.702,5.845,148.652
C09749=1203.785,98.581,-49.414,-178.705,5.844,148.653
C09750=1203.790,98.331,-49.396,-178.708,5.843,148.653
C09751=1203.795,98.082,-49.378,-178.710,5.842,148.654
C09752=1203.800,97.833,-49.359,-178.713,5.840,148.654
C09753=1203.805,97.584,-49.341,-178.715,5.840,148.655
C09754=1203.809,97.334,-49.322,-178.718,5.839,148.655
C09755=1203.814,97.085,-49.304,-178.721,5.838,148.656
C09756=1203.819,96.836,-49.285,-178.723,5.837,148.656
C09757=1203.824,96.587,-49.267,-178.726,5.836,148.657
C09758=1203.829,96.337,-49.249,-178.729,5.835,148.658
C09759=1203.834,96.088,-49.231,-178.731,5.834,148.658
C09760=1203.838,95.839,-49.212,-178.733,5.833,148.659
C09761=1203.844,95.590,-49.193,-178.736,5.831,148.659
C09762=1203.848,95.340,-49.175,-178.739,5.831,148.660
C09763=1203.853,95.091,-49.157,-178.741,5.830,148.660
C09764=1203.858,94.842,-49.139,-178.744,5.829,148.661
C09765=1203.863,94.593,-49.120,-178.746,5.828,148.661
C09766=1203.868,94.343,-49.101,-178.749,5.827,148.662
C09767=1203.873,94.094,-49.083,-178.752,5.826,148.663
C09768=1203.877,93.845,-49.066,-178.754,5.825,148.663
C09769=1203.882,93.595,-49.048,-178.757,5.824,148.664
C09770=1203.887,93.346,-49.030,-178.760,5.822,148.664
C09771=1203.892,93.096,-49.011,-178.762,5.822,148.665
C09772=1203.897,92.847,-48.993,-178.764,5.821,148.665
C09773=1203.902,92.598,-48.974,-178.767,5.819,148.666
C09774=1203.907,92.349,-48.956,-178.770,5.819,148.666
C09775=1203.912,92.100,-48.938,-178.772,5.818,148.667
C09776=1203.916,91.850,-48.920,-178.775,5.817,148.667
C09777=1203.921,91.601,-48.902,-178.778,5.816,148.668
C09778=1203.926,91.352,-48.884,-178.780,5.815,148.669
C09779=1203.931,91.103,-48.866,-178.783,5.813,148.669
C09780=1203.936,90.853,-48.848,-178.786,5.813,148.670
C09781=1203.941,90.604,-48.830,-178.788,5.812,148.670
C09782=1203.945,90.354,-48.811,-178.790,5.811,148.671
C09783=1203.950,90.105,-48.793,-178.793,5.810,148.671
C09784=1203.955,89.856,-48.775,-178.796,5.809,148.672
C09785=1203.960,89.607,-48.757,-178.798,5.808,148.672
C09786=1203.965,89.357,-48.739,-178.801,5.807,148.673
C09787=1203.970,89.108,-48.721,-178.804,5.806,148.673
C09788=1203.975,88.859,-48.703,-178.806,5.805,148.674
C09789=1203.979,88.609,-48.685,-178.809,5.804,148.675
C09790=1203.984,88.360,-48.667,-178.812,5.803,148.675
C09791=1203.989,88.111,-48.649,-178.814,5.802,148.676
C09792=1203.994,87.862,-48.631,-178.816,5.802,148.676
C09793=1203.999,87.612,-48.613,-178.819,5.800,148.677
C09794=1204.004,87.363,-48.595,-178.822,5.799,148.677
C09795=1204.009,87.113,-48.577,-178.824,5.799,148.678
C09796=1204.014,86.864,-48.559,-178.827,5.797,148.678
C09797=1204.019,86.615,-48.541,-178.830,5.796,148.679
C09798=1204.023,86.365,-48.523,-178.832,5.796,148.680
C09799=1204.028,86.116,-48.505,-178.834,5.795,148.680
C09800=1204.032,85.867,-48.488,-178.838,5.794,148.681
C09801=1204.037,85.618,-48.470,-178.840,5.793,148.681
C09802=1204.043,85.368,-48.452,-178.842,5.792,148.682
C09803=1204.047,85.119,-48.435,-178.845,5.791,148.683
C09804=1204.052,84.870,-48.417,-178.848,5.790,148.683
C09805=1204.057,84.621,-48.399,-178.850,5.789,148.684
C09806=1204.062,84.372,-48.381,-178.852,5.788,148.684
C09807=1204.067,84.122,-48.363,-178.856,5.787,148.685
C09808=1204.072,83.873,-48.345,-178.858,5.786,148.685
C09809=1204.077,83.623,-48.327,-178.860,5.785,148.686
C09810=1204.082,83.374,-48.309,-178.864,5.784,148.686
C09811=1204.087,83.124,-48.292,-178.866,5.783,148.687
C09812=1204.092,82.876,-48.275,-178.868,5.782,148.687
C09813=1204.096,82.626,-48.257,-178.871,5.782,148.688
C09814=1204.101,82.377,-48.239,-178.874,5.780,148.689
C09815=1204.107,82.127,-48.222,-178.876,5.780,148.689
C09816=1204.111,81.878,-48.204,-178.879,5.779,148.690
C09817=1204.116,81.629,-48.186,-178.881,5.778,148.690
C09818=1204.122,81.360,-48.167,-178.884,5.777,148.691
C09819=1204.127,81.092,-48.147,-178.887,5.776,148.692
C09820=1204.132,80.823,-48.129,-178.890,5.775,148.692
C09821=1204.137,80.555,-48.110,-178.893,5.774,148.693
C09822=1204.142,80.306,-48.092,-178.895,5.773,148.693
C09823=1204.147,80.056,-48.075,-178.898,5.772,148.694
C09824=1204.152,79.807,-48.057,-178.900,5.771,148.694
C09825=1204.157,79.557,-48.039,-178.903,5.770,148.695
C09826=1204.161,79.308,-48.022,-178.905,5.770,148.696
C09827=1204.166,79.059,-48.004,-178.908,5.768,148.696
C09828=1204.171,78.809,-47.987,-178.911,5.768,148.697
C09829=1204.176,78.560,-47.969,-178.913,5.767,148.697
C09830=1204.181,78.311,-47.952,-178.915,5.766,148.698
C09831=1204.186,78.062,-47.935,-178.919,5.765,148.698
C09832=1204.191,77.813,-47.917,-178.921,5.764,148.699
C09833=1204.196,77.563,-47.899,-178.923,5.763,148.700
C09834=1204.200,77.314,-47.882,-178.926,5.763,148.700
C09835=1204.206,77.065,-47.865,-178.928,5.762,148.701
C09836=1204.210,76.815,-47.847,-178.931,5.760,148.701
C09837=1204.216,76.566,-47.829,-178.934,5.760,148.702
C09838=1204.220,76.317,-47.812,-178.936,5.759,148.702
C09839=1204.225,76.067,-47.795,-178.939,5.758,148.703
C09840=1204.230,75.818,-47.777,-178.942,5.757,148.704
C09841=1204.234,75.568,-47.760,-178.944,5.756,148.704
C09842=1204.239,75.319,-47.742,-178.947,5.755,148.705
C09843=1204.245,75.069,-47.725,-178.949,5.755,148.705
C09844=1204.249,74.820,-47.708,-178.952,5.754,148.706
C09845=1204.255,74.571,-47.691,-178.955,5.753,148.707
C09846=1204.260,74.322,-47.673,-178.957,5.752,148.707
C09847=1204.264,74.073,-47.656,-178.960,5.751,148.708
C09848=1204.269,73.823,-47.639,-178.962,5.751,148.708
C09849=1204.274,73.573,-47.621,-178.965,5.749,148.709
C09850=1204.279,73.324,-47.604,-178.967,5.748,148.709
C09851=1204.284,73.074,-47.587,-178.970,5.748,148.710
C09852=1204.288,72.826,-47.569,-178.972,5.747,148.710
C09853=1204.294,72.577,-47.552,-178.975,5.746,148.711
C09854=1204.299,72.327,-47.535,-178.978,5.745,148.712
C09855=1204.303,72.078,-47.518,-178.980,5.744,148.712
C09856=1204.308,71.828,-47.501,-178.983,5.743,148.713
C09857=1204.313,71.579,-47.484,-178.985,5.743,148.714
C09858=1204.318,71.329,-47.466,-178.988,5.742,148.714
C09859=1204.323,71.080,-47.449,-178.991,5.741,148.715
C09860=1204.328,70.831,-47.432,-178.993,5.740,148.715
C09861=1204.333,70.582,-47.414,-178.996,5.739,148.716
C09862=1204.338,70.332,-47.398,-178.998,5.739,148.716
C09863=1204.343,70.082,-47.380,-179.001,5.738,148.717
C09864=1204.347,69.833,-47.364,-179.004,5.736,148.717
C09865=1204.352,69.584,-47.346,-179.006,5.736,148.718
C09866=1204.358,69.335,-47.329,-179.009,5.735,148.719
C09867=1204.362,69.085,-47.312,-179.011,5.734,148.719
C09868=1204.368,68.835,-47.295,-179.014,5.734,148.720
C09869=1204.372,68.586,-47.278,-179.017,5.732,148.721
C09870=1204.377,68.337,-47.260,-179.019,5.731,148.721
C09871=1204.382,68.088,-47.244,-179.022,5.731,148.722
C09872=1204.387,67.838,-47.227,-179.024,5.730,148.722
C09873=1204.392,67.589,-47.210,-179.026,5.729,148.723
C09874=1204.397,67.339,-47.192,-179.029,5.729,148.723
C09875=1204.401,67.090,-47.175,-179.032,5.727,148.724
C09876=1204.406,66.841,-47.159,-179.035,5.727,148.725
C09877=1204.412,66.591,-47.142,-179.037,5.726,148.725
C09878=1204.416,66.342,-47.125,-179.040,5.725,148.726
C09879=1204.421,66.092,-47.108,-179.042,5.725,148.726
C09880=1204.426,65.843,-47.092,-179.044,5.724,148.727
C09881=1204.431,65.594,-47.074,-179.048,5.723,148.728
C09882=1204.436,65.345,-47.057,-179.050,5.722,148.728
C09883=1204.441,65.095,-47.040,-179.052,5.721,148.729
C09884=1204.446,64.846,-47.023,-179.055,5.721,148.729
C09885=1204.450,64.597,-47.007,-179.058,5.720,148.730
C09886=1204.456,64.347,-46.989,-179.060,5.719,148.730
C09887=1204.460,64.097,-46.973,-179.063,5.718,148.731
C09888=1204.466,63.848,-46.956,-179.066,5.717,148.732
C09889=1204.470,63.599,-46.939,-179.068,5.716,148.732
C09890=1204.475,63.349,-46.923,-179.070,5.716,148.733
C09891=1204.481,63.100,-46.906,-179.073,5.715,148.733
C09892=1204.485,62.851,-46.889,-179.076,5.715,148.734
C09893=1204.490,62.601,-46.872,-179.078,5.713,148.735
C09894=1204.495,62.351,-46.855,-179.081,5.712,148.735
C09895=1204.500,62.103,-46.839,-179.084,5.712,148.736
C09896=1204.505,61.853,-46.821,-179.086,5.711,148.736
C09897=1204.510,61.603,-46.805,-179.088,5.710,148.737
C09898=1204.515,61.355,-46.789,-179.091,5.710,148.738
C09899=1204.520,61.105,-46.771,-179.093,5.709,148.738
C09900=1204.524,60.855,-46.755,-179.096,5.707,148.739
C09901=1204.530,60.606,-46.738,-179.099,5.707,148.739
C09902=1204.534,60.357,-46.722,-179.102,5.706,148.740
C09903=1204.539,60.107,-46.704,-179.104,5.705,148.741
C09904=1204.544,59.858,-46.688,-179.106,5.705,148.741
C09905=1204.549,59.609,-46.671,-179.109,5.704,148.742
C09906=1204.554,59.358,-46.655,-179.111,5.703,148.742
C09907=1204.559,59.110,-46.639,-179.114,5.702,148.743
C09908=1204.564,58.860,-46.622,-179.117,5.702,148.744
C09909=1204.568,58.611,-46.605,-179.120,5.701,148.744
C09910=1204.574,58.362,-46.588,-179.122,5.700,148.745
C09911=1204.579,58.112,-46.572,-179.124,5.700,148.745
C09912=1204.584,57.863,-46.555,-179.127,5.699,148.746
C09913=1204.589,57.613,-46.539,-179.129,5.698,148.746
C09914=1204.594,57.363,-46.522,-179.132,5.698,148.747
C09915=1204.599,57.115,-46.506,-179.135,5.696,148.748
C09916=1204.603,56.865,-46.489,-179.138,5.696,148.748
C09917=1204.608,56.616,-46.472,-179.140,5.695,148.749
C09918=1204.614,56.366,-46.456,-179.142,5.694,148.750
C09919=1204.618,56.117,-46.440,-179.145,5.694,148.750
C09920=1204.624,55.868,-46.423,-179.147,5.693,148.751
C09921=1204.628,55.618,-46.407,-179.150,5.692,148.751
C09922=1204.634,55.349,-46.389,-179.153,5.691,148.752
C09923=1204.639,55.081,-46.371,-179.156,5.690,148.753
C09924=1204.644,54.812,-46.354,-179.158,5.690,148.753
C09925=1204.650,54.545,-46.336,-179.161,5.689,148.754
C09926=1204.654,54.295,-46.319,-179.164,5.688,148.755
C09927=1204.660,54.045,-46.303,-179.166,5.687,148.755
C09928=1204.665,53.796,-46.287,-179.169,5.686,148.756
C09929=1204.669,53.546,-46.270,-179.172,5.686,148.756
C09930=1204.675,53.297,-46.254,-179.174,5.685,148.757
C09931=1204.679,53.048,-46.238,-179.176,5.684,148.758
C09932=1204.684,52.799,-46.221,-179.179,5.684,148.758
C09933=1204.689,52.549,-46.205,-179.182,5.683,148.759
C09934=1204.694,52.300,-46.189,-179.184,5.683,148.760
C09935=1204.699,52.050,-46.172,-179.186,5.682,148.760
C09936=1204.704,51.800,-46.156,-179.190,5.681,148.761
C09937=1204.709,51.551,-46.140,-179.192,5.680,148.761
C09938=1204.714,51.301,-46.124,-179.194,5.679,148.762
C09939=1204.719,51.052,-46.107,-179.197,5.679,148.762
C09940=1204.724,50.803,-46.091,-179.200,5.678,148.763
C09941=1204.729,50.553,-46.075,-179.202,5.677,148.764
C09942=1204.733,50.304,-46.058,-179.205,5.677,148.764
C09943=1204.739,50.055,-46.043,-179.207,5.676,148.765
C09944=1204.743,49.805,-46.026,-179.210,5.675,148.766
C09945=1204.749,49.556,-46.011,-179.212,5.675,148.766
C09946=1204.753,49.306,-45.994,-179.215,5.674,148.767
C09947=1204.758,49.057,-45.978,-179.217,5.673,148.767
C09948=1204.763,48.807,-45.962,-179.220,5.672,148.768
C09949=1204.768,48.558,-45.945,-179.223,5.672,148.769
C09950=1204.773,48.308,-45.929,-179.225,5.671,148.769
C09951=1204.778,48.060,-45.913,-179.228,5.670,148.770
C09952=1204.783,47.809,-45.897,-179.231,5.670,148.770
C09953=1204.788,47.561,-45.881,-179.233,5.669,148.771
C09954=1204.793,47.311,-45.865,-179.235,5.668,148.772
C09955=1204.798,47.061,-45.849,-179.238,5.668,148.772
C09956=1204.803,46.812,-45.833,-179.241,5.667,148.773
C09957=1204.808,46.562,-45.817,-179.243,5.667,148.774
C09958=1204.813,46.314,-45.801,-179.245,5.666,148.774
C09959=1204.818,46.063,-45.785,-179.248,5.665,148.775
C09960=1204.823,45.815,-45.769,-179.251,5.665,148.775
C09961=1204.828,45.565,-45.753,-179.253,5.664,148.776
C09962=1204.833,45.315,-45.737,-179.256,5.662,148.776
C09963=1204.838,45.066,-45.721,-179.259,5.662,148.777
C09964=1204.843,44.816,-45.705,-179.261,5.661,148.778
C09965=1204.848,44.567,-45.688,-179.264,5.661,148.778
C09966=1204.853,44.317,-45.672,-179.267,5.660,148.779
C09967=1204.858,44.068,-45.657,-179.269,5.659,148.780
C09968=1204.863,43.818,-45.640,-179.271,5.659,148.780
C09969=1204.868,43.569,-45.625,-179.274,5.658,148.781
C09970=1204.873,43.320,-45.610,-179.277,5.658,148.782
C09971=1204.877,43.071,-45.593,-179.279,5.657,148.782
C09972=1204.883,42.821,-45.577,-179.281,5.656,148.783
C09973=1204.888,42.572,-45.562,-179.284,5.656,148.783
C09974=1204.892,42.322,-45.545,-179.287,5.655,148.784
C09975=1204.898,42.073,-45.530,-179.289,5.654,148.785
C09976=1204.903,41.823,-45.514,-179.292,5.654,148.785
C09977=1204.908,41.573,-45.498,-179.294,5.653,148.786
C09978=1204.912,41.325,-45.482,-179.297,5.653,148.787
C09979=1204.917,41.075,-45.466,-179.299,5.652,148.787
C09980=1204.922,40.825,-45.451,-179.302,5.651,148.788
C09981=1204.928,40.576,-45.435,-179.304,5.651,148.788
C09982=1204.932,40.326,-45.418,-179.307,5.650,148.789
C09983=1204.938,40.077,-45.403,-179.310,5.649,148.790
C09984=1204.942,39.828,-45.388,-179.312,5.648,148.790
C09985=1204.947,39.578,-45.372,-179.315,5.647,148.791
C09986=1204.952,39.329,-45.356,-179.318,5.647,148.791
C09987=1204.958,39.080,-45.340,-179.320,5.646,148.792
C09988=1204.962,38.830,-45.324,-179.322,5.645,148.793
C09989=1204.967,38.580,-45.309,-179.325,5.645,148.793
C09990=1204.972,38.331,-45.294,-179.328,5.644,148.794
C09991=1204.977,38.081,-45.278,-179.330,5.644,148.795
C09992=1204.983,37.832,-45.262,-179.333,5.643,148.795
C09993=1204.987,37.583,-45.246,-179.335,5.642,148.796
C09994=1204.992,37.333,-45.230,-179.338,5.642,148.796
C09995=1204.997,37.084,-45.215,-179.340,5.641,148.797
C09996=1205.002,36.834,-45.199,-179.343,5.641,148.798
//INST
///DATE 2021/06/25 14:28
///ATTR SC,RW,RJ
////FRAME ROBOT
///GROUP1 RB1
NOP
MOVL C00000 V=800.0 PL=0
MOVL C00001 V=800.0 PL=0
MOVL C00002 V=800.0 PL=0
MOVL C00003 V=800.0 PL=0
MOVL C00004 V=800.0 PL=0
MOVL C00005 V=800.0 PL=0
MOVL C00006 V=800.0 PL=0
MOVL C00007 V=800.0 PL=0
MOVL C00008 V=800.0 PL=0
MOVL C00009 V=800.0 PL=0
MOVL C00010 V=800.0 PL=0
MOVL C00011 V=800.0 PL=0
MOVL C00012 V=800.0 PL=0
MOVL C00013 V=800.0 PL=0
MOVL C00014 V=800.0 PL=0
MOVL C00015 V=800.0 PL=0
MOVL C00016 V=800.0 PL=0
MOVL C00017 V=800.0 PL=0
MOVL C00018 V=800.0 PL=0
MOVL C00019 V=800.0 PL=0
MOVL C00020 V=800.0 PL=0
MOVL C00021 V=800.0 PL=0
MOVL C00022 V=800.0 PL=0
MOVL C00023 V=800.0 PL=0
MOVL C00024 V=800.0 PL=0
MOVL C00025 V=800.0 PL=0
MOVL C00026 V=800.0 PL=0
MOVL C00027 V=800.0 PL=0
MOVL C00028 V=800.0 PL=0
MOVL C00029 V=800.0 PL=0
MOVL C00030 V=800.0 PL=0
MOVL C00031 V=800.0 PL=0
MOVL C00032 V=800.0 PL=0
MOVL C00033 V=800.0 PL=0
MOVL C00034 V=800.0 PL=0
MOVL C00035 V=800.0 PL=0
MOVL C00036 V=800.0 PL=0
MOVL C00037 V=800.0 PL=0
MOVL C00038 V=800.0 PL=0
MOVL C00039 V=800.0 PL=0
MOVL C00040 V=800.0 PL=0
MOVL C00041 V=800.0 PL=0
MOVL C00042 V=800.0 PL=0
MOVL C00043 V=800.0 PL=0
MOVL C00044 V=800.0 PL=0
MOVL C00045 V=800.0 PL=0
MOVL C00046 V=800.0 PL=0
MOVL C00047 V=800.0 PL=0
MOVL C00048 V=800.0 PL=0
MOVL C00049 V=800.0 PL=0
MOVL C00050 V=800.0 PL=0
MOVL C00051 V=800.0 PL=0
MOVL C00052 V=800.0 PL=0
MOVL C00053 V=800.0 PL=0
MOVL C00054 V=800.0 PL=0
MOVL C00055 V=800.0 PL=0
MOVL C00056 V=800.0 PL=0
MOVL C00057 V=800.0 PL=0
MOVL C00058 V=800.0 PL=0
MOVL C00059 V=800.0 PL=0
MOVL C00060 V=800.0 PL=0
MOVL C00061 V=800.0 PL=0
MOVL C00062 V=800.0 PL=0
MOVL C00063 V=800.0 PL=0
MOVL C00064 V=800.0 PL=0
MOVL C00065 V=800.0 PL=0
MOVL C00066 V=800.0 PL=0
MOVL C00067 V=800.0 PL=0
MOVL C00068 V=800.0 PL=0
MOVL C00069 V=800.0 PL=0
MOVL C00070 V=800.0 PL=0
MOVL C00071 V=800.0 PL=0
MOVL C00072 V=800.0 PL=0
MOVL C00073 V=800.0 PL=0
MOVL C00074 V=800.0 PL=0
MOVL C00075 V=800.0 PL=0
MOVL C00076 V=800.0 PL=0
MOVL C00077 V=800.0 PL=0
MOVL C00078 V=800.0 PL=0
MOVL C00079 V=800.0 PL=0
MOVL C00080 V=800.0 PL=0
MOVL C00081 V=800.0 PL=0
MOVL C00082 V=800.0 PL=0
MOVL C00083 V=800.0 PL=0
MOVL C00084 V=800.0 PL=0
MOVL C00085 V=800.0 PL=0
MOVL C00086 V=800.0 PL=0
MOVL C00087 V=800.0 PL=0
MOVL C00088 V=800.0 PL=0
MOVL C00089 V=800.0 PL=0
MOVL C00090 V=800.0 PL=0
MOVL C00091 V=800.0 PL=0
MOVL C00092 V=800.0 PL=0
MOVL C00093 V=800.0 PL=0
MOVL C00094 V=800.0 PL=0
MOVL C00095 V=800.0 PL=0
MOVL C00096 V=800.0 PL=0
MOVL C00097 V=800.0 PL=0
MOVL C00098 V=800.0 PL=0
MOVL C00099 V=800.0 PL=0
MOVL C00100 V=800.0 PL=0
MOVL C00101 V=800.0 PL=0
MOVL C00102 V=800.0 PL=0
MOVL C00103 V=800.0 PL=0
MOVL C00104 V=800.0 PL=0
MOVL C00105 V=800.0 PL=0
MOVL C00106 V=800.0 PL=0
MOVL C00107 V=800.0 PL=0
MOVL C00108 V=800.0 PL=0
MOVL C00109 V=800.0 PL=0
MOVL C00110 V=800.0 PL=0
MOVL C00111 V=800.0 PL=0
MOVL C00112 V=800.0 PL=0
MOVL C00113 V=800.0 PL=0
MOVL C00114 V=800.0 PL=0
MOVL C00115 V=800.0 PL=0
MOVL C00116 V=800.0 PL=0
MOVL C00117 V=800.0 PL=0
MOVL C00118 V=800.0 PL=0
MOVL C00119 V=800.0 PL=0
MOVL C00120 V=800.0 PL=0
MOVL C00121 V=800.0 PL=0
MOVL C00122 V=800.0 PL=0
MOVL C00123 V=800.0 PL=0
MOVL C00124 V=800.0 PL=0
MOVL C00125 V=800.0 PL=0
MOVL C00126 V=800.0 PL=0
MOVL C00127 V=800.0 PL=0
MOVL C00128 V=800.0 PL=0
MOVL C00129 V=800.0 PL=0
MOVL C00130 V=800.0 PL=0
MOVL C00131 V=800.0 PL=0
MOVL C00132 V=800.0 PL=0
MOVL C00133 V=800.0 PL=0
MOVL C00134 V=800.0 PL=0
MOVL C00135 V=800.0 PL=0
MOVL C00136 V=800.0 PL=0
MOVL C00137 V=800.0 PL=0
MOVL C00138 V=800.0 PL=0
MOVL C00139 V=800.0 PL=0
MOVL C00140 V=800.0 PL=0
MOVL C00141 V=800.0 PL=0
MOVL C00142 V=800.0 PL=0
MOVL C00143 V=800.0 PL=0
MOVL C00144 V=800.0 PL=0
MOVL C00145 V=800.0 PL=0
MOVL C00146 V=800.0 PL=0
MOVL C00147 V=800.0 PL=0
MOVL C00148 V=800.0 PL=0
MOVL C00149 V=800.0 PL=0
MOVL C00150 V=800.0 PL=0
MOVL C00151 V=800.0 PL=0
MOVL C00152 V=800.0 PL=0
MOVL C00153 V=800.0 PL=0
MOVL C00154 V=800.0 PL=0
MOVL C00155 V=800.0 PL=0
MOVL C00156 V=800.0 PL=0
MOVL C00157 V=800.0 PL=0
MOVL C00158 V=800.0 PL=0
MOVL C00159 V=800.0 PL=0
MOVL C00160 V=800.0 PL=0
MOVL C00161 V=800.0 PL=0
MOVL C00162 V=800.0 PL=0
MOVL C00163 V=800.0 PL=0
MOVL C00164 V=800.0 PL=0
MOVL C00165 V=800.0 PL=0
MOVL C00166 V=800.0 PL=0
MOVL C00167 V=800.0 PL=0
MOVL C00168 V=800.0 PL=0
MOVL C00169 V=800.0 PL=0
MOVL C00170 V=800.0 PL=0
MOVL C00171 V=800.0 PL=0
MOVL C00172 V=800.0 PL=0
MOVL C00173 V=800.0 PL=0
MOVL C00174 V=800.0 PL=0
MOVL C00175 V=800.0 PL=0
MOVL C00176 V=800.0 PL=0
MOVL C00177 V=800.0 PL=0
MOVL C00178 V=800.0 PL=0
MOVL C00179 V=800.0 PL=0
MOVL C00180 V=800.0 PL=0
MOVL C00181 V=800.0 PL=0
MOVL C00182 V=800.0 PL=0
MOVL C00183 V=800.0 PL=0
MOVL C00184 V=800.0 PL=0
MOVL C00185 V=800.0 PL=0
MOVL C00186 V=800.0 PL=0
MOVL C00187 V=800.0 PL=0
MOVL C00188 V=800.0 PL=0
MOVL C00189 V=800.0 PL=0
MOVL C00190 V=800.0 PL=0
MOVL C00191 V=800.0 PL=0
MOVL C00192 V=800.0 PL=0
MOVL C00193 V=800.0 PL=0
MOVL C00194 V=800.0 PL=0
MOVL C00195 V=800.0 PL=0
MOVL C00196 V=800.0 PL=0
MOVL C00197 V=800.0 PL=0
MOVL C00198 V=800.0 PL=0
MOVL C00199 V=800.0 PL=0
MOVL C00200 V=800.0 PL=0
MOVL C00201 V=800.0 PL=0
MOVL C00202 V=800.0 PL=0
MOVL C00203 V=800.0 PL=0
MOVL C00204 V=800.0 PL=0
MOVL C00205 V=800.0 PL=0
MOVL C00206 V=800.0 PL=0
MOVL C00207 V=800.0 PL=0
MOVL C00208 V=800.0 PL=0
MOVL C00209 V=800.0 PL=0
MOVL C00210 V=800.0 PL=0
MOVL C00211 V=800.0 PL=0
MOVL C00212 V=800.0 PL=0
MOVL C00213 V=800.0 PL=0
MOVL C00214 V=800.0 PL=0
MOVL C00215 V=800.0 PL=0
MOVL C00216 V=800.0 PL=0
MOVL C00217 V=800.0 PL=0
MOVL C00218 V=800.0 PL=0
MOVL C00219 V=800.0 PL=0
MOVL C00220 V=800.0 PL=0
MOVL C00221 V=800.0 PL=0
MOVL C00222 V=800.0 PL=0
MOVL C00223 V=800.0 PL=0
MOVL C00224 V=800.0 PL=0
MOVL C00225 V=800.0 PL=0
MOVL C00226 V=800.0 PL=0
MOVL C00227 V=800.0 PL=0
MOVL C00228 V=800.0 PL=0
MOVL C00229 V=800.0 PL=0
MOVL C00230 V=800.0 PL=0
MOVL C00231 V=800.0 PL=0
MOVL C00232 V=800.0 PL=0
MOVL C00233 V=800.0 PL=0
MOVL C00234 V=800.0 PL=0
MOVL C00235 V=800.0 PL=0
MOVL C00236 V=800.0 PL=0
MOVL C00237 V=800.0 PL=0
MOVL C00238 V=800.0 PL=0
MOVL C00239 V=800.0 PL=0
MOVL C00240 V=800.0 PL=0
MOVL C00241 V=800.0 PL=0
MOVL C00242 V=800.0 PL=0
MOVL C00243 V=800.0 PL=0
MOVL C00244 V=800.0 PL=0
MOVL C00245 V=800.0 PL=0
MOVL C00246 V=800.0 PL=0
MOVL C00247 V=800.0 PL=0
MOVL C00248 V=800.0 PL=0
MOVL C00249 V=800.0 PL=0
MOVL C00250 V=800.0 PL=0
MOVL C00251 V=800.0 PL=0
MOVL C00252 V=800.0 PL=0
MOVL C00253 V=800.0 PL=0
MOVL C00254 V=800.0 PL=0
MOVL C00255 V=800.0 PL=0
MOVL C00256 V=800.0 PL=0
MOVL C00257 V=800.0 PL=0
MOVL C00258 V=800.0 PL=0
MOVL C00259 V=800.0 PL=0
MOVL C00260 V=800.0 PL=0
MOVL C00261 V=800.0 PL=0
MOVL C00262 V=800.0 PL=0
MOVL C00263 V=800.0 PL=0
MOVL C00264 V=800.0 PL=0
MOVL C00265 V=800.0 PL=0
MOVL C00266 V=800.0 PL=0
MOVL C00267 V=800.0 PL=0
MOVL C00268 V=800.0 PL=0
MOVL C00269 V=800.0 PL=0
MOVL C00270 V=800.0 PL=0
MOVL C00271 V=800.0 PL=0
MOVL C00272 V=800.0 PL=0
MOVL C00273 V=800.0 PL=0
MOVL C00274 V=800.0 PL=0
MOVL C00275 V=800.0 PL=0
MOVL C00276 V=800.0 PL=0
MOVL C00277 V=800.0 PL=0
MOVL C00278 V=800.0 PL=0
MOVL C00279 V=800.0 PL=0
MOVL C00280 V=800.0 PL=0
MOVL C00281 V=800.0 PL=0
MOVL C00282 V=800.0 PL=0
MOVL C00283 V=800.0 PL=0
MOVL C00284 V=800.0 PL=0
MOVL C00285 V=800.0 PL=0
MOVL C00286 V=800.0 PL=0
MOVL C00287 V=800.0 PL=0
MOVL C00288 V=800.0 PL=0
MOVL C00289 V=800.0 PL=0
MOVL C00290 V=800.0 PL=0
MOVL C00291 V=800.0 PL=0
MOVL C00292 V=800.0 PL=0
MOVL C00293 V=800.0 PL=0
MOVL C00294 V=800.0 PL=0
MOVL C00295 V=800.0 PL=0
MOVL C00296 V=800.0 PL=0
MOVL C00297 V=800.0 PL=0
MOVL C00298 V=800.0 PL=0
MOVL C00299 V=800.0 PL=0
MOVL C00300 V=800.0 PL=0
MOVL C00301 V=800.0 PL=0
MOVL C00302 V=800.0 PL=0
MOVL C00303 V=800.0 PL=0
MOVL C00304 V=800.0 PL=0
MOVL C00305 V=800.0 PL=0
MOVL C00306 V=800.0 PL=0
MOVL C00307 V=800.0 PL=0
MOVL C00308 V=800.0 PL=0
MOVL C00309 V=800.0 PL=0
MOVL C00310 V=800.0 PL=0
MOVL C00311 V=800.0 PL=0
MOVL C00312 V=800.0 PL=0
MOVL C00313 V=800.0 PL=0
MOVL C00314 V=800.0 PL=0
MOVL C00315 V=800.0 PL=0
MOVL C00316 V=800.0 PL=0
MOVL C00317 V=800.0 PL=0
MOVL C00318 V=800.0 PL=0
MOVL C00319 V=800.0 PL=0
MOVL C00320 V=800.0 PL=0
MOVL C00321 V=800.0 PL=0
MOVL C00322 V=800.0 PL=0
MOVL C00323 V=800.0 PL=0
MOVL C00324 V=800.0 PL=0
MOVL C00325 V=800.0 PL=0
MOVL C00326 V=800.0 PL=0
MOVL C00327 V=800.0 PL=0
MOVL C00328 V=800.0 PL=0
MOVL C00329 V=800.0 PL=0
MOVL C00330 V=800.0 PL=0
MOVL C00331 V=800.0 PL=0
MOVL C00332 V=800.0 PL=0
MOVL C00333 V=800.0 PL=0
MOVL C00334 V=800.0 PL=0
MOVL C00335 V=800.0 PL=0
MOVL C00336 V=800.0 PL=0
MOVL C00337 V=800.0 PL=0
MOVL C00338 V=800.0 PL=0
MOVL C00339 V=800.0 PL=0
MOVL C00340 V=800.0 PL=0
MOVL C00341 V=800.0 PL=0
MOVL C00342 V=800.0 PL=0
MOVL C00343 V=800.0 PL=0
MOVL C00344 V=800.0 PL=0
MOVL C00345 V=800.0 PL=0
MOVL C00346 V=800.0 PL=0
MOVL C00347 V=800.0 PL=0
MOVL C00348 V=800.0 PL=0
MOVL C00349 V=800.0 PL=0
MOVL C00350 V=800.0 PL=0
MOVL C00351 V=800.0 PL=0
MOVL C00352 V=800.0 PL=0
MOVL C00353 V=800.0 PL=0
MOVL C00354 V=800.0 PL=0
MOVL C00355 V=800.0 PL=0
MOVL C00356 V=800.0 PL=0
MOVL C00357 V=800.0 PL=0
MOVL C00358 V=800.0 PL=0
MOVL C00359 V=800.0 PL=0
MOVL C00360 V=800.0 PL=0
MOVL C00361 V=800.0 PL=0
MOVL C00362 V=800.0 PL=0
MOVL C00363 V=800.0 PL=0
MOVL C00364 V=800.0 PL=0
MOVL C00365 V=800.0 PL=0
MOVL C00366 V=800.0 PL=0
MOVL C00367 V=800.0 PL=0
MOVL C00368 V=800.0 PL=0
MOVL C00369 V=800.0 PL=0
MOVL C00370 V=800.0 PL=0
MOVL C00371 V=800.0 PL=0
MOVL C00372 V=800.0 PL=0
MOVL C00373 V=800.0 PL=0
MOVL C00374 V=800.0 PL=0
MOVL C00375 V=800.0 PL=0
MOVL C00376 V=800.0 PL=0
MOVL C00377 V=800.0 PL=0
MOVL C00378 V=800.0 PL=0
MOVL C00379 V=800.0 PL=0
MOVL C00380 V=800.0 PL=0
MOVL C00381 V=800.0 PL=0
MOVL C00382 V=800.0 PL=0
MOVL C00383 V=800.0 PL=0
MOVL C00384 V=800.0 PL=0
MOVL C00385 V=800.0 PL=0
MOVL C00386 V=800.0 PL=0
MOVL C00387 V=800.0 PL=0
MOVL C00388 V=800.0 PL=0
MOVL C00389 V=800.0 PL=0
MOVL C00390 V=800.0 PL=0
MOVL C00391 V=800.0 PL=0
MOVL C00392 V=800.0 PL=0
MOVL C00393 V=800.0 PL=0
MOVL C00394 V=800.0 PL=0
MOVL C00395 V=800.0 PL=0
MOVL C00396 V=800.0 PL=0
MOVL C00397 V=800.0 PL=0
MOVL C00398 V=800.0 PL=0
MOVL C00399 V=800.0 PL=0
MOVL C00400 V=800.0 PL=0
MOVL C00401 V=800.0 PL=0
MOVL C00402 V=800.0 PL=0
MOVL C00403 V=800.0 PL=0
MOVL C00404 V=800.0 PL=0
MOVL C00405 V=800.0 PL=0
MOVL C00406 V=800.0 PL=0
MOVL C00407 V=800.0 PL=0
MOVL C00408 V=800.0 PL=0
MOVL C00409 V=800.0 PL=0
MOVL C00410 V=800.0 PL=0
MOVL C00411 V=800.0 PL=0
MOVL C00412 V=800.0 PL=0
MOVL C00413 V=800.0 PL=0
MOVL C00414 V=800.0 PL=0
MOVL C00415 V=800.0 PL=0
MOVL C00416 V=800.0 PL=0
MOVL C00417 V=800.0 PL=0
MOVL C00418 V=800.0 PL=0
MOVL C00419 V=800.0 PL=0
MOVL C00420 V=800.0 PL=0
MOVL C00421 V=800.0 PL=0
MOVL C00422 V=800.0 PL=0
MOVL C00423 V=800.0 PL=0
MOVL C00424 V=800.0 PL=0
MOVL C00425 V=800.0 PL=0
MOVL C00426 V=800.0 PL=0
MOVL C00427 V=800.0 PL=0
MOVL C00428 V=800.0 PL=0
MOVL C00429 V=800.0 PL=0
MOVL C00430 V=800.0 PL=0
MOVL C00431 V=800.0 PL=0
MOVL C00432 V=800.0 PL=0
MOVL C00433 V=800.0 PL=0
MOVL C00434 V=800.0 PL=0
MOVL C00435 V=800.0 PL=0
MOVL C00436 V=800.0 PL=0
MOVL C00437 V=800.0 PL=0
MOVL C00438 V=800.0 PL=0
MOVL C00439 V=800.0 PL=0
MOVL C00440 V=800.0 PL=0
MOVL C00441 V=800.0 PL=0
MOVL C00442 V=800.0 PL=0
MOVL C00443 V=800.0 PL=0
MOVL C00444 V=800.0 PL=0
MOVL C00445 V=800.0 PL=0
MOVL C00446 V=800.0 PL=0
MOVL C00447 V=800.0 PL=0
MOVL C00448 V=800.0 PL=0
MOVL C00449 V=800.0 PL=0
MOVL C00450 V=800.0 PL=0
MOVL C00451 V=800.0 PL=0
MOVL C00452 V=800.0 PL=0
MOVL C00453 V=800.0 PL=0
MOVL C00454 V=800.0 PL=0
MOVL C00455 V=800.0 PL=0
MOVL C00456 V=800.0 PL=0
MOVL C00457 V=800.0 PL=0
MOVL C00458 V=800.0 PL=0
MOVL C00459 V=800.0 PL=0
MOVL C00460 V=800.0 PL=0
MOVL C00461 V=800.0 PL=0
MOVL C00462 V=800.0 PL=0
MOVL C00463 V=800.0 PL=0
MOVL C00464 V=800.0 PL=0
MOVL C00465 V=800.0 PL=0
MOVL C00466 V=800.0 PL=0
MOVL C00467 V=800.0 PL=0
MOVL C00468 V=800.0 PL=0
MOVL C00469 V=800.0 PL=0
MOVL C00470 V=800.0 PL=0
MOVL C00471 V=800.0 PL=0
MOVL C00472 V=800.0 PL=0
MOVL C00473 V=800.0 PL=0
MOVL C00474 V=800.0 PL=0
MOVL C00475 V=800.0 PL=0
MOVL C00476 V=800.0 PL=0
MOVL C00477 V=800.0 PL=0
MOVL C00478 V=800.0 PL=0
MOVL C00479 V=800.0 PL=0
MOVL C00480 V=800.0 PL=0
MOVL C00481 V=800.0 PL=0
MOVL C00482 V=800.0 PL=0
MOVL C00483 V=800.0 PL=0
MOVL C00484 V=800.0 PL=0
MOVL C00485 V=800.0 PL=0
MOVL C00486 V=800.0 PL=0
MOVL C00487 V=800.0 PL=0
MOVL C00488 V=800.0 PL=0
MOVL C00489 V=800.0 PL=0
MOVL C00490 V=800.0 PL=0
MOVL C00491 V=800.0 PL=0
MOVL C00492 V=800.0 PL=0
MOVL C00493 V=800.0 PL=0
MOVL C00494 V=800.0 PL=0
MOVL C00495 V=800.0 PL=0
MOVL C00496 V=800.0 PL=0
MOVL C00497 V=800.0 PL=0
MOVL C00498 V=800.0 PL=0
MOVL C00499 V=800.0 PL=0
MOVL C00500 V=800.0 PL=0
MOVL C00501 V=800.0 PL=0
MOVL C00502 V=800.0 PL=0
MOVL C00503 V=800.0 PL=0
MOVL C00504 V=800.0 PL=0
MOVL C00505 V=800.0 PL=0
MOVL C00506 V=800.0 PL=0
MOVL C00507 V=800.0 PL=0
MOVL C00508 V=800.0 PL=0
MOVL C00509 V=800.0 PL=0
MOVL C00510 V=800.0 PL=0
MOVL C00511 V=800.0 PL=0
MOVL C00512 V=800.0 PL=0
MOVL C00513 V=800.0 PL=0
MOVL C00514 V=800.0 PL=0
MOVL C00515 V=800.0 PL=0
MOVL C00516 V=800.0 PL=0
MOVL C00517 V=800.0 PL=0
MOVL C00518 V=800.0 PL=0
MOVL C00519 V=800.0 PL=0
MOVL C00520 V=800.0 PL=0
MOVL C00521 V=800.0 PL=0
MOVL C00522 V=800.0 PL=0
MOVL C00523 V=800.0 PL=0
MOVL C00524 V=800.0 PL=0
MOVL C00525 V=800.0 PL=0
MOVL C00526 V=800.0 PL=0
MOVL C00527 V=800.0 PL=0
MOVL C00528 V=800.0 PL=0
MOVL C00529 V=800.0 PL=0
MOVL C00530 V=800.0 PL=0
MOVL C00531 V=800.0 PL=0
MOVL C00532 V=800.0 PL=0
MOVL C00533 V=800.0 PL=0
MOVL C00534 V=800.0 PL=0
MOVL C00535 V=800.0 PL=0
MOVL C00536 V=800.0 PL=0
MOVL C00537 V=800.0 PL=0
MOVL C00538 V=800.0 PL=0
MOVL C00539 V=800.0 PL=0
MOVL C00540 V=800.0 PL=0
MOVL C00541 V=800.0 PL=0
MOVL C00542 V=800.0 PL=0
MOVL C00543 V=800.0 PL=0
MOVL C00544 V=800.0 PL=0
MOVL C00545 V=800.0 PL=0
MOVL C00546 V=800.0 PL=0
MOVL C00547 V=800.0 PL=0
MOVL C00548 V=800.0 PL=0
MOVL C00549 V=800.0 PL=0
MOVL C00550 V=800.0 PL=0
MOVL C00551 V=800.0 PL=0
MOVL C00552 V=800.0 PL=0
MOVL C00553 V=800.0 PL=0
MOVL C00554 V=800.0 PL=0
MOVL C00555 V=800.0 PL=0
MOVL C00556 V=800.0 PL=0
MOVL C00557 V=800.0 PL=0
MOVL C00558 V=800.0 PL=0
MOVL C00559 V=800.0 PL=0
MOVL C00560 V=800.0 PL=0
MOVL C00561 V=800.0 PL=0
MOVL C00562 V=800.0 PL=0
MOVL C00563 V=800.0 PL=0
MOVL C00564 V=800.0 PL=0
MOVL C00565 V=800.0 PL=0
MOVL C00566 V=800.0 PL=0
MOVL C00567 V=800.0 PL=0
MOVL C00568 V=800.0 PL=0
MOVL C00569 V=800.0 PL=0
MOVL C00570 V=800.0 PL=0
MOVL C00571 V=800.0 PL=0
MOVL C00572 V=800.0 PL=0
MOVL C00573 V=800.0 PL=0
MOVL C00574 V=800.0 PL=0
MOVL C00575 V=800.0 PL=0
MOVL C00576 V=800.0 PL=0
MOVL C00577 V=800.0 PL=0
MOVL C00578 V=800.0 PL=0
MOVL C00579 V=800.0 PL=0
MOVL C00580 V=800.0 PL=0
MOVL C00581 V=800.0 PL=0
MOVL C00582 V=800.0 PL=0
MOVL C00583 V=800.0 PL=0
MOVL C00584 V=800.0 PL=0
MOVL C00585 V=800.0 PL=0
MOVL C00586 V=800.0 PL=0
MOVL C00587 V=800.0 PL=0
MOVL C00588 V=800.0 PL=0
MOVL C00589 V=800.0 PL=0
MOVL C00590 V=800.0 PL=0
MOVL C00591 V=800.0 PL=0
MOVL C00592 V=800.0 PL=0
MOVL C00593 V=800.0 PL=0
MOVL C00594 V=800.0 PL=0
MOVL C00595 V=800.0 PL=0
MOVL C00596 V=800.0 PL=0
MOVL C00597 V=800.0 PL=0
MOVL C00598 V=800.0 PL=0
MOVL C00599 V=800.0 PL=0
MOVL C00600 V=800.0 PL=0
MOVL C00601 V=800.0 PL=0
MOVL C00602 V=800.0 PL=0
MOVL C00603 V=800.0 PL=0
MOVL C00604 V=800.0 PL=0
MOVL C00605 V=800.0 PL=0
MOVL C00606 V=800.0 PL=0
MOVL C00607 V=800.0 PL=0
MOVL C00608 V=800.0 PL=0
MOVL C00609 V=800.0 PL=0
MOVL C00610 V=800.0 PL=0
MOVL C00611 V=800.0 PL=0
MOVL C00612 V=800.0 PL=0
MOVL C00613 V=800.0 PL=0
MOVL C00614 V=800.0 PL=0
MOVL C00615 V=800.0 PL=0
MOVL C00616 V=800.0 PL=0
MOVL C00617 V=800.0 PL=0
MOVL C00618 V=800.0 PL=0
MOVL C00619 V=800.0 PL=0
MOVL C00620 V=800.0 PL=0
MOVL C00621 V=800.0 PL=0
MOVL C00622 V=800.0 PL=0
MOVL C00623 V=800.0 PL=0
MOVL C00624 V=800.0 PL=0
MOVL C00625 V=800.0 PL=0
MOVL C00626 V=800.0 PL=0
MOVL C00627 V=800.0 PL=0
MOVL C00628 V=800.0 PL=0
MOVL C00629 V=800.0 PL=0
MOVL C00630 V=800.0 PL=0
MOVL C00631 V=800.0 PL=0
MOVL C00632 V=800.0 PL=0
MOVL C00633 V=800.0 PL=0
MOVL C00634 V=800.0 PL=0
MOVL C00635 V=800.0 PL=0
MOVL C00636 V=800.0 PL=0
MOVL C00637 V=800.0 PL=0
MOVL C00638 V=800.0 PL=0
MOVL C00639 V=800.0 PL=0
MOVL C00640 V=800.0 PL=0
MOVL C00641 V=800.0 PL=0
MOVL C00642 V=800.0 PL=0
MOVL C00643 V=800.0 PL=0
MOVL C00644 V=800.0 PL=0
MOVL C00645 V=800.0 PL=0
MOVL C00646 V=800.0 PL=0
MOVL C00647 V=800.0 PL=0
MOVL C00648 V=800.0 PL=0
MOVL C00649 V=800.0 PL=0
MOVL C00650 V=800.0 PL=0
MOVL C00651 V=800.0 PL=0
MOVL C00652 V=800.0 PL=0
MOVL C00653 V=800.0 PL=0
MOVL C00654 V=800.0 PL=0
MOVL C00655 V=800.0 PL=0
MOVL C00656 V=800.0 PL=0
MOVL C00657 V=800.0 PL=0
MOVL C00658 V=800.0 PL=0
MOVL C00659 V=800.0 PL=0
MOVL C00660 V=800.0 PL=0
MOVL C00661 V=800.0 PL=0
MOVL C00662 V=800.0 PL=0
MOVL C00663 V=800.0 PL=0
MOVL C00664 V=800.0 PL=0
MOVL C00665 V=800.0 PL=0
MOVL C00666 V=800.0 PL=0
MOVL C00667 V=800.0 PL=0
MOVL C00668 V=800.0 PL=0
MOVL C00669 V=800.0 PL=0
MOVL C00670 V=800.0 PL=0
MOVL C00671 V=800.0 PL=0
MOVL C00672 V=800.0 PL=0
MOVL C00673 V=800.0 PL=0
MOVL C00674 V=800.0 PL=0
MOVL C00675 V=800.0 PL=0
MOVL C00676 V=800.0 PL=0
MOVL C00677 V=800.0 PL=0
MOVL C00678 V=800.0 PL=0
MOVL C00679 V=800.0 PL=0
MOVL C00680 V=800.0 PL=0
MOVL C00681 V=800.0 PL=0
MOVL C00682 V=800.0 PL=0
MOVL C00683 V=800.0 PL=0
MOVL C00684 V=800.0 PL=0
MOVL C00685 V=800.0 PL=0
MOVL C00686 V=800.0 PL=0
MOVL C00687 V=800.0 PL=0
MOVL C00688 V=800.0 PL=0
MOVL C00689 V=800.0 PL=0
MOVL C00690 V=800.0 PL=0
MOVL C00691 V=800.0 PL=0
MOVL C00692 V=800.0 PL=0
MOVL C00693 V=800.0 PL=0
MOVL C00694 V=800.0 PL=0
MOVL C00695 V=800.0 PL=0
MOVL C00696 V=800.0 PL=0
MOVL C00697 V=800.0 PL=0
MOVL C00698 V=800.0 PL=0
MOVL C00699 V=800.0 PL=0
MOVL C00700 V=800.0 PL=0
MOVL C00701 V=800.0 PL=0
MOVL C00702 V=800.0 PL=0
MOVL C00703 V=800.0 PL=0
MOVL C00704 V=800.0 PL=0
MOVL C00705 V=800.0 PL=0
MOVL C00706 V=800.0 PL=0
MOVL C00707 V=800.0 PL=0
MOVL C00708 V=800.0 PL=0
MOVL C00709 V=800.0 PL=0
MOVL C00710 V=800.0 PL=0
MOVL C00711 V=800.0 PL=0
MOVL C00712 V=800.0 PL=0
MOVL C00713 V=800.0 PL=0
MOVL C00714 V=800.0 PL=0
MOVL C00715 V=800.0 PL=0
MOVL C00716 V=800.0 PL=0
MOVL C00717 V=800.0 PL=0
MOVL C00718 V=800.0 PL=0
MOVL C00719 V=800.0 PL=0
MOVL C00720 V=800.0 PL=0
MOVL C00721 V=800.0 PL=0
MOVL C00722 V=800.0 PL=0
MOVL C00723 V=800.0 PL=0
MOVL C00724 V=800.0 PL=0
MOVL C00725 V=800.0 PL=0
MOVL C00726 V=800.0 PL=0
MOVL C00727 V=800.0 PL=0
MOVL C00728 V=800.0 PL=0
MOVL C00729 V=800.0 PL=0
MOVL C00730 V=800.0 PL=0
MOVL C00731 V=800.0 PL=0
MOVL C00732 V=800.0 PL=0
MOVL C00733 V=800.0 PL=0
MOVL C00734 V=800.0 PL=0
MOVL C00735 V=800.0 PL=0
MOVL C00736 V=800.0 PL=0
MOVL C00737 V=800.0 PL=0
MOVL C00738 V=800.0 PL=0
MOVL C00739 V=800.0 PL=0
MOVL C00740 V=800.0 PL=0
MOVL C00741 V=800.0 PL=0
MOVL C00742 V=800.0 PL=0
MOVL C00743 V=800.0 PL=0
MOVL C00744 V=800.0 PL=0
MOVL C00745 V=800.0 PL=0
MOVL C00746 V=800.0 PL=0
MOVL C00747 V=800.0 PL=0
MOVL C00748 V=800.0 PL=0
MOVL C00749 V=800.0 PL=0
MOVL C00750 V=800.0 PL=0
MOVL C00751 V=800.0 PL=0
MOVL C00752 V=800.0 PL=0
MOVL C00753 V=800.0 PL=0
MOVL C00754 V=800.0 PL=0
MOVL C00755 V=800.0 PL=0
MOVL C00756 V=800.0 PL=0
MOVL C00757 V=800.0 PL=0
MOVL C00758 V=800.0 PL=0
MOVL C00759 V=800.0 PL=0
MOVL C00760 V=800.0 PL=0
MOVL C00761 V=800.0 PL=0
MOVL C00762 V=800.0 PL=0
MOVL C00763 V=800.0 PL=0
MOVL C00764 V=800.0 PL=0
MOVL C00765 V=800.0 PL=0
MOVL C00766 V=800.0 PL=0
MOVL C00767 V=800.0 PL=0
MOVL C00768 V=800.0 PL=0
MOVL C00769 V=800.0 PL=0
MOVL C00770 V=800.0 PL=0
MOVL C00771 V=800.0 PL=0
MOVL C00772 V=800.0 PL=0
MOVL C00773 V=800.0 PL=0
MOVL C00774 V=800.0 PL=0
MOVL C00775 V=800.0 PL=0
MOVL C00776 V=800.0 PL=0
MOVL C00777 V=800.0 PL=0
MOVL C00778 V=800.0 PL=0
MOVL C00779 V=800.0 PL=0
MOVL C00780 V=800.0 PL=0
MOVL C00781 V=800.0 PL=0
MOVL C00782 V=800.0 PL=0
MOVL C00783 V=800.0 PL=0
MOVL C00784 V=800.0 PL=0
MOVL C00785 V=800.0 PL=0
MOVL C00786 V=800.0 PL=0
MOVL C00787 V=800.0 PL=0
MOVL C00788 V=800.0 PL=0
MOVL C00789 V=800.0 PL=0
MOVL C00790 V=800.0 PL=0
MOVL C00791 V=800.0 PL=0
MOVL C00792 V=800.0 PL=0
MOVL C00793 V=800.0 PL=0
MOVL C00794 V=800.0 PL=0
MOVL C00795 V=800.0 PL=0
MOVL C00796 V=800.0 PL=0
MOVL C00797 V=800.0 PL=0
MOVL C00798 V=800.0 PL=0
MOVL C00799 V=800.0 PL=0
MOVL C00800 V=800.0 PL=0
MOVL C00801 V=800.0 PL=0
MOVL C00802 V=800.0 PL=0
MOVL C00803 V=800.0 PL=0
MOVL C00804 V=800.0 PL=0
MOVL C00805 V=800.0 PL=0
MOVL C00806 V=800.0 PL=0
MOVL C00807 V=800.0 PL=0
MOVL C00808 V=800.0 PL=0
MOVL C00809 V=800.0 PL=0
MOVL C00810 V=800.0 PL=0
MOVL C00811 V=800.0 PL=0
MOVL C00812 V=800.0 PL=0
MOVL C00813 V=800.0 PL=0
MOVL C00814 V=800.0 PL=0
MOVL C00815 V=800.0 PL=0
MOVL C00816 V=800.0 PL=0
MOVL C00817 V=800.0 PL=0
MOVL C00818 V=800.0 PL=0
MOVL C00819 V=800.0 PL=0
MOVL C00820 V=800.0 PL=0
MOVL C00821 V=800.0 PL=0
MOVL C00822 V=800.0 PL=0
MOVL C00823 V=800.0 PL=0
MOVL C00824 V=800.0 PL=0
MOVL C00825 V=800.0 PL=0
MOVL C00826 V=800.0 PL=0
MOVL C00827 V=800.0 PL=0
MOVL C00828 V=800.0 PL=0
MOVL C00829 V=800.0 PL=0
MOVL C00830 V=800.0 PL=0
MOVL C00831 V=800.0 PL=0
MOVL C00832 V=800.0 PL=0
MOVL C00833 V=800.0 PL=0
MOVL C00834 V=800.0 PL=0
MOVL C00835 V=800.0 PL=0
MOVL C00836 V=800.0 PL=0
MOVL C00837 V=800.0 PL=0
MOVL C00838 V=800.0 PL=0
MOVL C00839 V=800.0 PL=0
MOVL C00840 V=800.0 PL=0
MOVL C00841 V=800.0 PL=0
MOVL C00842 V=800.0 PL=0
MOVL C00843 V=800.0 PL=0
MOVL C00844 V=800.0 PL=0
MOVL C00845 V=800.0 PL=0
MOVL C00846 V=800.0 PL=0
MOVL C00847 V=800.0 PL=0
MOVL C00848 V=800.0 PL=0
MOVL C00849 V=800.0 PL=0
MOVL C00850 V=800.0 PL=0
MOVL C00851 V=800.0 PL=0
MOVL C00852 V=800.0 PL=0
MOVL C00853 V=800.0 PL=0
MOVL C00854 V=800.0 PL=0
MOVL C00855 V=800.0 PL=0
MOVL C00856 V=800.0 PL=0
MOVL C00857 V=800.0 PL=0
MOVL C00858 V=800.0 PL=0
MOVL C00859 V=800.0 PL=0
MOVL C00860 V=800.0 PL=0
MOVL C00861 V=800.0 PL=0
MOVL C00862 V=800.0 PL=0
MOVL C00863 V=800.0 PL=0
MOVL C00864 V=800.0 PL=0
MOVL C00865 V=800.0 PL=0
MOVL C00866 V=800.0 PL=0
MOVL C00867 V=800.0 PL=0
MOVL C00868 V=800.0 PL=0
MOVL C00869 V=800.0 PL=0
MOVL C00870 V=800.0 PL=0
MOVL C00871 V=800.0 PL=0
MOVL C00872 V=800.0 PL=0
MOVL C00873 V=800.0 PL=0
MOVL C00874 V=800.0 PL=0
MOVL C00875 V=800.0 PL=0
MOVL C00876 V=800.0 PL=0
MOVL C00877 V=800.0 PL=0
MOVL C00878 V=800.0 PL=0
MOVL C00879 V=800.0 PL=0
MOVL C00880 V=800.0 PL=0
MOVL C00881 V=800.0 PL=0
MOVL C00882 V=800.0 PL=0
MOVL C00883 V=800.0 PL=0
MOVL C00884 V=800.0 PL=0
MOVL C00885 V=800.0 PL=0
MOVL C00886 V=800.0 PL=0
MOVL C00887 V=800.0 PL=0
MOVL C00888 V=800.0 PL=0
MOVL C00889 V=800.0 PL=0
MOVL C00890 V=800.0 PL=0
MOVL C00891 V=800.0 PL=0
MOVL C00892 V=800.0 PL=0
MOVL C00893 V=800.0 PL=0
MOVL C00894 V=800.0 PL=0
MOVL C00895 V=800.0 PL=0
MOVL C00896 V=800.0 PL=0
MOVL C00897 V=800.0 PL=0
MOVL C00898 V=800.0 PL=0
MOVL C00899 V=800.0 PL=0
MOVL C00900 V=800.0 PL=0
MOVL C00901 V=800.0 PL=0
MOVL C00902 V=800.0 PL=0
MOVL C00903 V=800.0 PL=0
MOVL C00904 V=800.0 PL=0
MOVL C00905 V=800.0 PL=0
MOVL C00906 V=800.0 PL=0
MOVL C00907 V=800.0 PL=0
MOVL C00908 V=800.0 PL=0
MOVL C00909 V=800.0 PL=0
MOVL C00910 V=800.0 PL=0
MOVL C00911 V=800.0 PL=0
MOVL C00912 V=800.0 PL=0
MOVL C00913 V=800.0 PL=0
MOVL C00914 V=800.0 PL=0
MOVL C00915 V=800.0 PL=0
MOVL C00916 V=800.0 PL=0
MOVL C00917 V=800.0 PL=0
MOVL C00918 V=800.0 PL=0
MOVL C00919 V=800.0 PL=0
MOVL C00920 V=800.0 PL=0
MOVL C00921 V=800.0 PL=0
MOVL C00922 V=800.0 PL=0
MOVL C00923 V=800.0 PL=0
MOVL C00924 V=800.0 PL=0
MOVL C00925 V=800.0 PL=0
MOVL C00926 V=800.0 PL=0
MOVL C00927 V=800.0 PL=0
MOVL C00928 V=800.0 PL=0
MOVL C00929 V=800.0 PL=0
MOVL C00930 V=800.0 PL=0
MOVL C00931 V=800.0 PL=0
MOVL C00932 V=800.0 PL=0
MOVL C00933 V=800.0 PL=0
MOVL C00934 V=800.0 PL=0
MOVL C00935 V=800.0 PL=0
MOVL C00936 V=800.0 PL=0
MOVL C00937 V=800.0 PL=0
MOVL C00938 V=800.0 PL=0
MOVL C00939 V=800.0 PL=0
MOVL C00940 V=800.0 PL=0
MOVL C00941 V=800.0 PL=0
MOVL C00942 V=800.0 PL=0
MOVL C00943 V=800.0 PL=0
MOVL C00944 V=800.0 PL=0
MOVL C00945 V=800.0 PL=0
MOVL C00946 V=800.0 PL=0
MOVL C00947 V=800.0 PL=0
MOVL C00948 V=800.0 PL=0
MOVL C00949 V=800.0 PL=0
MOVL C00950 V=800.0 PL=0
MOVL C00951 V=800.0 PL=0
MOVL C00952 V=800.0 PL=0
MOVL C00953 V=800.0 PL=0
MOVL C00954 V=800.0 PL=0
MOVL C00955 V=800.0 PL=0
MOVL C00956 V=800.0 PL=0
MOVL C00957 V=800.0 PL=0
MOVL C00958 V=800.0 PL=0
MOVL C00959 V=800.0 PL=0
MOVL C00960 V=800.0 PL=0
MOVL C00961 V=800.0 PL=0
MOVL C00962 V=800.0 PL=0
MOVL C00963 V=800.0 PL=0
MOVL C00964 V=800.0 PL=0
MOVL C00965 V=800.0 PL=0
MOVL C00966 V=800.0 PL=0
MOVL C00967 V=800.0 PL=0
MOVL C00968 V=800.0 PL=0
MOVL C00969 V=800.0 PL=0
MOVL C00970 V=800.0 PL=0
MOVL C00971 V=800.0 PL=0
MOVL C00972 V=800.0 PL=0
MOVL C00973 V=800.0 PL=0
MOVL C00974 V=800.0 PL=0
MOVL C00975 V=800.0 PL=0
MOVL C00976 V=800.0 PL=0
MOVL C00977 V=800.0 PL=0
MOVL C00978 V=800.0 PL=0
MOVL C00979 V=800.0 PL=0
MOVL C00980 V=800.0 PL=0
MOVL C00981 V=800.0 PL=0
MOVL C00982 V=800.0 PL=0
MOVL C00983 V=800.0 PL=0
MOVL C00984 V=800.0 PL=0
MOVL C00985 V=800.0 PL=0
MOVL C00986 V=800.0 PL=0
MOVL C00987 V=800.0 PL=0
MOVL C00988 V=800.0 PL=0
MOVL C00989 V=800.0 PL=0
MOVL C00990 V=800.0 PL=0
MOVL C00991 V=800.0 PL=0
MOVL C00992 V=800.0 PL=0
MOVL C00993 V=800.0 PL=0
MOVL C00994 V=800.0 PL=0
MOVL C00995 V=800.0 PL=0
MOVL C00996 V=800.0 PL=0
MOVL C00997 V=800.0 PL=0
MOVL C00998 V=800.0 PL=0
MOVL C00999 V=800.0 PL=0
MOVL C01000 V=800.0 PL=0
MOVL C01001 V=800.0 PL=0
MOVL C01002 V=800.0 PL=0
MOVL C01003 V=800.0 PL=0
MOVL C01004 V=800.0 PL=0
MOVL C01005 V=800.0 PL=0
MOVL C01006 V=800.0 PL=0
MOVL C01007 V=800.0 PL=0
MOVL C01008 V=800.0 PL=0
MOVL C01009 V=800.0 PL=0
MOVL C01010 V=800.0 PL=0
MOVL C01011 V=800.0 PL=0
MOVL C01012 V=800.0 PL=0
MOVL C01013 V=800.0 PL=0
MOVL C01014 V=800.0 PL=0
MOVL C01015 V=800.0 PL=0
MOVL C01016 V=800.0 PL=0
MOVL C01017 V=800.0 PL=0
MOVL C01018 V=800.0 PL=0
MOVL C01019 V=800.0 PL=0
MOVL C01020 V=800.0 PL=0
MOVL C01021 V=800.0 PL=0
MOVL C01022 V=800.0 PL=0
MOVL C01023 V=800.0 PL=0
MOVL C01024 V=800.0 PL=0
MOVL C01025 V=800.0 PL=0
MOVL C01026 V=800.0 PL=0
MOVL C01027 V=800.0 PL=0
MOVL C01028 V=800.0 PL=0
MOVL C01029 V=800.0 PL=0
MOVL C01030 V=800.0 PL=0
MOVL C01031 V=800.0 PL=0
MOVL C01032 V=800.0 PL=0
MOVL C01033 V=800.0 PL=0
MOVL C01034 V=800.0 PL=0
MOVL C01035 V=800.0 PL=0
MOVL C01036 V=800.0 PL=0
MOVL C01037 V=800.0 PL=0
MOVL C01038 V=800.0 PL=0
MOVL C01039 V=800.0 PL=0
MOVL C01040 V=800.0 PL=0
MOVL C01041 V=800.0 PL=0
MOVL C01042 V=800.0 PL=0
MOVL C01043 V=800.0 PL=0
MOVL C01044 V=800.0 PL=0
MOVL C01045 V=800.0 PL=0
MOVL C01046 V=800.0 PL=0
MOVL C01047 V=800.0 PL=0
MOVL C01048 V=800.0 PL=0
MOVL C01049 V=800.0 PL=0
MOVL C01050 V=800.0 PL=0
MOVL C01051 V=800.0 PL=0
MOVL C01052 V=800.0 PL=0
MOVL C01053 V=800.0 PL=0
MOVL C01054 V=800.0 PL=0
MOVL C01055 V=800.0 PL=0
MOVL C01056 V=800.0 PL=0
MOVL C01057 V=800.0 PL=0
MOVL C01058 V=800.0 PL=0
MOVL C01059 V=800.0 PL=0
MOVL C01060 V=800.0 PL=0
MOVL C01061 V=800.0 PL=0
MOVL C01062 V=800.0 PL=0
MOVL C01063 V=800.0 PL=0
MOVL C01064 V=800.0 PL=0
MOVL C01065 V=800.0 PL=0
MOVL C01066 V=800.0 PL=0
MOVL C01067 V=800.0 PL=0
MOVL C01068 V=800.0 PL=0
MOVL C01069 V=800.0 PL=0
MOVL C01070 V=800.0 PL=0
MOVL C01071 V=800.0 PL=0
MOVL C01072 V=800.0 PL=0
MOVL C01073 V=800.0 PL=0
MOVL C01074 V=800.0 PL=0
MOVL C01075 V=800.0 PL=0
MOVL C01076 V=800.0 PL=0
MOVL C01077 V=800.0 PL=0
MOVL C01078 V=800.0 PL=0
MOVL C01079 V=800.0 PL=0
MOVL C01080 V=800.0 PL=0
MOVL C01081 V=800.0 PL=0
MOVL C01082 V=800.0 PL=0
MOVL C01083 V=800.0 PL=0
MOVL C01084 V=800.0 PL=0
MOVL C01085 V=800.0 PL=0
MOVL C01086 V=800.0 PL=0
MOVL C01087 V=800.0 PL=0
MOVL C01088 V=800.0 PL=0
MOVL C01089 V=800.0 PL=0
MOVL C01090 V=800.0 PL=0
MOVL C01091 V=800.0 PL=0
MOVL C01092 V=800.0 PL=0
MOVL C01093 V=800.0 PL=0
MOVL C01094 V=800.0 PL=0
MOVL C01095 V=800.0 PL=0
MOVL C01096 V=800.0 PL=0
MOVL C01097 V=800.0 PL=0
MOVL C01098 V=800.0 PL=0
MOVL C01099 V=800.0 PL=0
MOVL C01100 V=800.0 PL=0
MOVL C01101 V=800.0 PL=0
MOVL C01102 V=800.0 PL=0
MOVL C01103 V=800.0 PL=0
MOVL C01104 V=800.0 PL=0
MOVL C01105 V=800.0 PL=0
MOVL C01106 V=800.0 PL=0
MOVL C01107 V=800.0 PL=0
MOVL C01108 V=800.0 PL=0
MOVL C01109 V=800.0 PL=0
MOVL C01110 V=800.0 PL=0
MOVL C01111 V=800.0 PL=0
MOVL C01112 V=800.0 PL=0
MOVL C01113 V=800.0 PL=0
MOVL C01114 V=800.0 PL=0
MOVL C01115 V=800.0 PL=0
MOVL C01116 V=800.0 PL=0
MOVL C01117 V=800.0 PL=0
MOVL C01118 V=800.0 PL=0
MOVL C01119 V=800.0 PL=0
MOVL C01120 V=800.0 PL=0
MOVL C01121 V=800.0 PL=0
MOVL C01122 V=800.0 PL=0
MOVL C01123 V=800.0 PL=0
MOVL C01124 V=800.0 PL=0
MOVL C01125 V=800.0 PL=0
MOVL C01126 V=800.0 PL=0
MOVL C01127 V=800.0 PL=0
MOVL C01128 V=800.0 PL=0
MOVL C01129 V=800.0 PL=0
MOVL C01130 V=800.0 PL=0
MOVL C01131 V=800.0 PL=0
MOVL C01132 V=800.0 PL=0
MOVL C01133 V=800.0 PL=0
MOVL C01134 V=800.0 PL=0
MOVL C01135 V=800.0 PL=0
MOVL C01136 V=800.0 PL=0
MOVL C01137 V=800.0 PL=0
MOVL C01138 V=800.0 PL=0
MOVL C01139 V=800.0 PL=0
MOVL C01140 V=800.0 PL=0
MOVL C01141 V=800.0 PL=0
MOVL C01142 V=800.0 PL=0
MOVL C01143 V=800.0 PL=0
MOVL C01144 V=800.0 PL=0
MOVL C01145 V=800.0 PL=0
MOVL C01146 V=800.0 PL=0
MOVL C01147 V=800.0 PL=0
MOVL C01148 V=800.0 PL=0
MOVL C01149 V=800.0 PL=0
MOVL C01150 V=800.0 PL=0
MOVL C01151 V=800.0 PL=0
MOVL C01152 V=800.0 PL=0
MOVL C01153 V=800.0 PL=0
MOVL C01154 V=800.0 PL=0
MOVL C01155 V=800.0 PL=0
MOVL C01156 V=800.0 PL=0
MOVL C01157 V=800.0 PL=0
MOVL C01158 V=800.0 PL=0
MOVL C01159 V=800.0 PL=0
MOVL C01160 V=800.0 PL=0
MOVL C01161 V=800.0 PL=0
MOVL C01162 V=800.0 PL=0
MOVL C01163 V=800.0 PL=0
MOVL C01164 V=800.0 PL=0
MOVL C01165 V=800.0 PL=0
MOVL C01166 V=800.0 PL=0
MOVL C01167 V=800.0 PL=0
MOVL C01168 V=800.0 PL=0
MOVL C01169 V=800.0 PL=0
MOVL C01170 V=800.0 PL=0
MOVL C01171 V=800.0 PL=0
MOVL C01172 V=800.0 PL=0
MOVL C01173 V=800.0 PL=0
MOVL C01174 V=800.0 PL=0
MOVL C01175 V=800.0 PL=0
MOVL C01176 V=800.0 PL=0
MOVL C01177 V=800.0 PL=0
MOVL C01178 V=800.0 PL=0
MOVL C01179 V=800.0 PL=0
MOVL C01180 V=800.0 PL=0
MOVL C01181 V=800.0 PL=0
MOVL C01182 V=800.0 PL=0
MOVL C01183 V=800.0 PL=0
MOVL C01184 V=800.0 PL=0
MOVL C01185 V=800.0 PL=0
MOVL C01186 V=800.0 PL=0
MOVL C01187 V=800.0 PL=0
MOVL C01188 V=800.0 PL=0
MOVL C01189 V=800.0 PL=0
MOVL C01190 V=800.0 PL=0
MOVL C01191 V=800.0 PL=0
MOVL C01192 V=800.0 PL=0
MOVL C01193 V=800.0 PL=0
MOVL C01194 V=800.0 PL=0
MOVL C01195 V=800.0 PL=0
MOVL C01196 V=800.0 PL=0
MOVL C01197 V=800.0 PL=0
MOVL C01198 V=800.0 PL=0
MOVL C01199 V=800.0 PL=0
MOVL C01200 V=800.0 PL=0
MOVL C01201 V=800.0 PL=0
MOVL C01202 V=800.0 PL=0
MOVL C01203 V=800.0 PL=0
MOVL C01204 V=800.0 PL=0
MOVL C01205 V=800.0 PL=0
MOVL C01206 V=800.0 PL=0
MOVL C01207 V=800.0 PL=0
MOVL C01208 V=800.0 PL=0
MOVL C01209 V=800.0 PL=0
MOVL C01210 V=800.0 PL=0
MOVL C01211 V=800.0 PL=0
MOVL C01212 V=800.0 PL=0
MOVL C01213 V=800.0 PL=0
MOVL C01214 V=800.0 PL=0
MOVL C01215 V=800.0 PL=0
MOVL C01216 V=800.0 PL=0
MOVL C01217 V=800.0 PL=0
MOVL C01218 V=800.0 PL=0
MOVL C01219 V=800.0 PL=0
MOVL C01220 V=800.0 PL=0
MOVL C01221 V=800.0 PL=0
MOVL C01222 V=800.0 PL=0
MOVL C01223 V=800.0 PL=0
MOVL C01224 V=800.0 PL=0
MOVL C01225 V=800.0 PL=0
MOVL C01226 V=800.0 PL=0
MOVL C01227 V=800.0 PL=0
MOVL C01228 V=800.0 PL=0
MOVL C01229 V=800.0 PL=0
MOVL C01230 V=800.0 PL=0
MOVL C01231 V=800.0 PL=0
MOVL C01232 V=800.0 PL=0
MOVL C01233 V=800.0 PL=0
MOVL C01234 V=800.0 PL=0
MOVL C01235 V=800.0 PL=0
MOVL C01236 V=800.0 PL=0
MOVL C01237 V=800.0 PL=0
MOVL C01238 V=800.0 PL=0
MOVL C01239 V=800.0 PL=0
MOVL C01240 V=800.0 PL=0
MOVL C01241 V=800.0 PL=0
MOVL C01242 V=800.0 PL=0
MOVL C01243 V=800.0 PL=0
MOVL C01244 V=800.0 PL=0
MOVL C01245 V=800.0 PL=0
MOVL C01246 V=800.0 PL=0
MOVL C01247 V=800.0 PL=0
MOVL C01248 V=800.0 PL=0
MOVL C01249 V=800.0 PL=0
MOVL C01250 V=800.0 PL=0
MOVL C01251 V=800.0 PL=0
MOVL C01252 V=800.0 PL=0
MOVL C01253 V=800.0 PL=0
MOVL C01254 V=800.0 PL=0
MOVL C01255 V=800.0 PL=0
MOVL C01256 V=800.0 PL=0
MOVL C01257 V=800.0 PL=0
MOVL C01258 V=800.0 PL=0
MOVL C01259 V=800.0 PL=0
MOVL C01260 V=800.0 PL=0
MOVL C01261 V=800.0 PL=0
MOVL C01262 V=800.0 PL=0
MOVL C01263 V=800.0 PL=0
MOVL C01264 V=800.0 PL=0
MOVL C01265 V=800.0 PL=0
MOVL C01266 V=800.0 PL=0
MOVL C01267 V=800.0 PL=0
MOVL C01268 V=800.0 PL=0
MOVL C01269 V=800.0 PL=0
MOVL C01270 V=800.0 PL=0
MOVL C01271 V=800.0 PL=0
MOVL C01272 V=800.0 PL=0
MOVL C01273 V=800.0 PL=0
MOVL C01274 V=800.0 PL=0
MOVL C01275 V=800.0 PL=0
MOVL C01276 V=800.0 PL=0
MOVL C01277 V=800.0 PL=0
MOVL C01278 V=800.0 PL=0
MOVL C01279 V=800.0 PL=0
MOVL C01280 V=800.0 PL=0
MOVL C01281 V=800.0 PL=0
MOVL C01282 V=800.0 PL=0
MOVL C01283 V=800.0 PL=0
MOVL C01284 V=800.0 PL=0
MOVL C01285 V=800.0 PL=0
MOVL C01286 V=800.0 PL=0
MOVL C01287 V=800.0 PL=0
MOVL C01288 V=800.0 PL=0
MOVL C01289 V=800.0 PL=0
MOVL C01290 V=800.0 PL=0
MOVL C01291 V=800.0 PL=0
MOVL C01292 V=800.0 PL=0
MOVL C01293 V=800.0 PL=0
MOVL C01294 V=800.0 PL=0
MOVL C01295 V=800.0 PL=0
MOVL C01296 V=800.0 PL=0
MOVL C01297 V=800.0 PL=0
MOVL C01298 V=800.0 PL=0
MOVL C01299 V=800.0 PL=0
MOVL C01300 V=800.0 PL=0
MOVL C01301 V=800.0 PL=0
MOVL C01302 V=800.0 PL=0
MOVL C01303 V=800.0 PL=0
MOVL C01304 V=800.0 PL=0
MOVL C01305 V=800.0 PL=0
MOVL C01306 V=800.0 PL=0
MOVL C01307 V=800.0 PL=0
MOVL C01308 V=800.0 PL=0
MOVL C01309 V=800.0 PL=0
MOVL C01310 V=800.0 PL=0
MOVL C01311 V=800.0 PL=0
MOVL C01312 V=800.0 PL=0
MOVL C01313 V=800.0 PL=0
MOVL C01314 V=800.0 PL=0
MOVL C01315 V=800.0 PL=0
MOVL C01316 V=800.0 PL=0
MOVL C01317 V=800.0 PL=0
MOVL C01318 V=800.0 PL=0
MOVL C01319 V=800.0 PL=0
MOVL C01320 V=800.0 PL=0
MOVL C01321 V=800.0 PL=0
MOVL C01322 V=800.0 PL=0
MOVL C01323 V=800.0 PL=0
MOVL C01324 V=800.0 PL=0
MOVL C01325 V=800.0 PL=0
MOVL C01326 V=800.0 PL=0
MOVL C01327 V=800.0 PL=0
MOVL C01328 V=800.0 PL=0
MOVL C01329 V=800.0 PL=0
MOVL C01330 V=800.0 PL=0
MOVL C01331 V=800.0 PL=0
MOVL C01332 V=800.0 PL=0
MOVL C01333 V=800.0 PL=0
MOVL C01334 V=800.0 PL=0
MOVL C01335 V=800.0 PL=0
MOVL C01336 V=800.0 PL=0
MOVL C01337 V=800.0 PL=0
MOVL C01338 V=800.0 PL=0
MOVL C01339 V=800.0 PL=0
MOVL C01340 V=800.0 PL=0
MOVL C01341 V=800.0 PL=0
MOVL C01342 V=800.0 PL=0
MOVL C01343 V=800.0 PL=0
MOVL C01344 V=800.0 PL=0
MOVL C01345 V=800.0 PL=0
MOVL C01346 V=800.0 PL=0
MOVL C01347 V=800.0 PL=0
MOVL C01348 V=800.0 PL=0
MOVL C01349 V=800.0 PL=0
MOVL C01350 V=800.0 PL=0
MOVL C01351 V=800.0 PL=0
MOVL C01352 V=800.0 PL=0
MOVL C01353 V=800.0 PL=0
MOVL C01354 V=800.0 PL=0
MOVL C01355 V=800.0 PL=0
MOVL C01356 V=800.0 PL=0
MOVL C01357 V=800.0 PL=0
MOVL C01358 V=800.0 PL=0
MOVL C01359 V=800.0 PL=0
MOVL C01360 V=800.0 PL=0
MOVL C01361 V=800.0 PL=0
MOVL C01362 V=800.0 PL=0
MOVL C01363 V=800.0 PL=0
MOVL C01364 V=800.0 PL=0
MOVL C01365 V=800.0 PL=0
MOVL C01366 V=800.0 PL=0
MOVL C01367 V=800.0 PL=0
MOVL C01368 V=800.0 PL=0
MOVL C01369 V=800.0 PL=0
MOVL C01370 V=800.0 PL=0
MOVL C01371 V=800.0 PL=0
MOVL C01372 V=800.0 PL=0
MOVL C01373 V=800.0 PL=0
MOVL C01374 V=800.0 PL=0
MOVL C01375 V=800.0 PL=0
MOVL C01376 V=800.0 PL=0
MOVL C01377 V=800.0 PL=0
MOVL C01378 V=800.0 PL=0
MOVL C01379 V=800.0 PL=0
MOVL C01380 V=800.0 PL=0
MOVL C01381 V=800.0 PL=0
MOVL C01382 V=800.0 PL=0
MOVL C01383 V=800.0 PL=0
MOVL C01384 V=800.0 PL=0
MOVL C01385 V=800.0 PL=0
MOVL C01386 V=800.0 PL=0
MOVL C01387 V=800.0 PL=0
MOVL C01388 V=800.0 PL=0
MOVL C01389 V=800.0 PL=0
MOVL C01390 V=800.0 PL=0
MOVL C01391 V=800.0 PL=0
MOVL C01392 V=800.0 PL=0
MOVL C01393 V=800.0 PL=0
MOVL C01394 V=800.0 PL=0
MOVL C01395 V=800.0 PL=0
MOVL C01396 V=800.0 PL=0
MOVL C01397 V=800.0 PL=0
MOVL C01398 V=800.0 PL=0
MOVL C01399 V=800.0 PL=0
MOVL C01400 V=800.0 PL=0
MOVL C01401 V=800.0 PL=0
MOVL C01402 V=800.0 PL=0
MOVL C01403 V=800.0 PL=0
MOVL C01404 V=800.0 PL=0
MOVL C01405 V=800.0 PL=0
MOVL C01406 V=800.0 PL=0
MOVL C01407 V=800.0 PL=0
MOVL C01408 V=800.0 PL=0
MOVL C01409 V=800.0 PL=0
MOVL C01410 V=800.0 PL=0
MOVL C01411 V=800.0 PL=0
MOVL C01412 V=800.0 PL=0
MOVL C01413 V=800.0 PL=0
MOVL C01414 V=800.0 PL=0
MOVL C01415 V=800.0 PL=0
MOVL C01416 V=800.0 PL=0
MOVL C01417 V=800.0 PL=0
MOVL C01418 V=800.0 PL=0
MOVL C01419 V=800.0 PL=0
MOVL C01420 V=800.0 PL=0
MOVL C01421 V=800.0 PL=0
MOVL C01422 V=800.0 PL=0
MOVL C01423 V=800.0 PL=0
MOVL C01424 V=800.0 PL=0
MOVL C01425 V=800.0 PL=0
MOVL C01426 V=800.0 PL=0
MOVL C01427 V=800.0 PL=0
MOVL C01428 V=800.0 PL=0
MOVL C01429 V=800.0 PL=0
MOVL C01430 V=800.0 PL=0
MOVL C01431 V=800.0 PL=0
MOVL C01432 V=800.0 PL=0
MOVL C01433 V=800.0 PL=0
MOVL C01434 V=800.0 PL=0
MOVL C01435 V=800.0 PL=0
MOVL C01436 V=800.0 PL=0
MOVL C01437 V=800.0 PL=0
MOVL C01438 V=800.0 PL=0
MOVL C01439 V=800.0 PL=0
MOVL C01440 V=800.0 PL=0
MOVL C01441 V=800.0 PL=0
MOVL C01442 V=800.0 PL=0
MOVL C01443 V=800.0 PL=0
MOVL C01444 V=800.0 PL=0
MOVL C01445 V=800.0 PL=0
MOVL C01446 V=800.0 PL=0
MOVL C01447 V=800.0 PL=0
MOVL C01448 V=800.0 PL=0
MOVL C01449 V=800.0 PL=0
MOVL C01450 V=800.0 PL=0
MOVL C01451 V=800.0 PL=0
MOVL C01452 V=800.0 PL=0
MOVL C01453 V=800.0 PL=0
MOVL C01454 V=800.0 PL=0
MOVL C01455 V=800.0 PL=0
MOVL C01456 V=800.0 PL=0
MOVL C01457 V=800.0 PL=0
MOVL C01458 V=800.0 PL=0
MOVL C01459 V=800.0 PL=0
MOVL C01460 V=800.0 PL=0
MOVL C01461 V=800.0 PL=0
MOVL C01462 V=800.0 PL=0
MOVL C01463 V=800.0 PL=0
MOVL C01464 V=800.0 PL=0
MOVL C01465 V=800.0 PL=0
MOVL C01466 V=800.0 PL=0
MOVL C01467 V=800.0 PL=0
MOVL C01468 V=800.0 PL=0
MOVL C01469 V=800.0 PL=0
MOVL C01470 V=800.0 PL=0
MOVL C01471 V=800.0 PL=0
MOVL C01472 V=800.0 PL=0
MOVL C01473 V=800.0 PL=0
MOVL C01474 V=800.0 PL=0
MOVL C01475 V=800.0 PL=0
MOVL C01476 V=800.0 PL=0
MOVL C01477 V=800.0 PL=0
MOVL C01478 V=800.0 PL=0
MOVL C01479 V=800.0 PL=0
MOVL C01480 V=800.0 PL=0
MOVL C01481 V=800.0 PL=0
MOVL C01482 V=800.0 PL=0
MOVL C01483 V=800.0 PL=0
MOVL C01484 V=800.0 PL=0
MOVL C01485 V=800.0 PL=0
MOVL C01486 V=800.0 PL=0
MOVL C01487 V=800.0 PL=0
MOVL C01488 V=800.0 PL=0
MOVL C01489 V=800.0 PL=0
MOVL C01490 V=800.0 PL=0
MOVL C01491 V=800.0 PL=0
MOVL C01492 V=800.0 PL=0
MOVL C01493 V=800.0 PL=0
MOVL C01494 V=800.0 PL=0
MOVL C01495 V=800.0 PL=0
MOVL C01496 V=800.0 PL=0
MOVL C01497 V=800.0 PL=0
MOVL C01498 V=800.0 PL=0
MOVL C01499 V=800.0 PL=0
MOVL C01500 V=800.0 PL=0
MOVL C01501 V=800.0 PL=0
MOVL C01502 V=800.0 PL=0
MOVL C01503 V=800.0 PL=0
MOVL C01504 V=800.0 PL=0
MOVL C01505 V=800.0 PL=0
MOVL C01506 V=800.0 PL=0
MOVL C01507 V=800.0 PL=0
MOVL C01508 V=800.0 PL=0
MOVL C01509 V=800.0 PL=0
MOVL C01510 V=800.0 PL=0
MOVL C01511 V=800.0 PL=0
MOVL C01512 V=800.0 PL=0
MOVL C01513 V=800.0 PL=0
MOVL C01514 V=800.0 PL=0
MOVL C01515 V=800.0 PL=0
MOVL C01516 V=800.0 PL=0
MOVL C01517 V=800.0 PL=0
MOVL C01518 V=800.0 PL=0
MOVL C01519 V=800.0 PL=0
MOVL C01520 V=800.0 PL=0
MOVL C01521 V=800.0 PL=0
MOVL C01522 V=800.0 PL=0
MOVL C01523 V=800.0 PL=0
MOVL C01524 V=800.0 PL=0
MOVL C01525 V=800.0 PL=0
MOVL C01526 V=800.0 PL=0
MOVL C01527 V=800.0 PL=0
MOVL C01528 V=800.0 PL=0
MOVL C01529 V=800.0 PL=0
MOVL C01530 V=800.0 PL=0
MOVL C01531 V=800.0 PL=0
MOVL C01532 V=800.0 PL=0
MOVL C01533 V=800.0 PL=0
MOVL C01534 V=800.0 PL=0
MOVL C01535 V=800.0 PL=0
MOVL C01536 V=800.0 PL=0
MOVL C01537 V=800.0 PL=0
MOVL C01538 V=800.0 PL=0
MOVL C01539 V=800.0 PL=0
MOVL C01540 V=800.0 PL=0
MOVL C01541 V=800.0 PL=0
MOVL C01542 V=800.0 PL=0
MOVL C01543 V=800.0 PL=0
MOVL C01544 V=800.0 PL=0
MOVL C01545 V=800.0 PL=0
MOVL C01546 V=800.0 PL=0
MOVL C01547 V=800.0 PL=0
MOVL C01548 V=800.0 PL=0
MOVL C01549 V=800.0 PL=0
MOVL C01550 V=800.0 PL=0
MOVL C01551 V=800.0 PL=0
MOVL C01552 V=800.0 PL=0
MOVL C01553 V=800.0 PL=0
MOVL C01554 V=800.0 PL=0
MOVL C01555 V=800.0 PL=0
MOVL C01556 V=800.0 PL=0
MOVL C01557 V=800.0 PL=0
MOVL C01558 V=800.0 PL=0
MOVL C01559 V=800.0 PL=0
MOVL C01560 V=800.0 PL=0
MOVL C01561 V=800.0 PL=0
MOVL C01562 V=800.0 PL=0
MOVL C01563 V=800.0 PL=0
MOVL C01564 V=800.0 PL=0
MOVL C01565 V=800.0 PL=0
MOVL C01566 V=800.0 PL=0
MOVL C01567 V=800.0 PL=0
MOVL C01568 V=800.0 PL=0
MOVL C01569 V=800.0 PL=0
MOVL C01570 V=800.0 PL=0
MOVL C01571 V=800.0 PL=0
MOVL C01572 V=800.0 PL=0
MOVL C01573 V=800.0 PL=0
MOVL C01574 V=800.0 PL=0
MOVL C01575 V=800.0 PL=0
MOVL C01576 V=800.0 PL=0
MOVL C01577 V=800.0 PL=0
MOVL C01578 V=800.0 PL=0
MOVL C01579 V=800.0 PL=0
MOVL C01580 V=800.0 PL=0
MOVL C01581 V=800.0 PL=0
MOVL C01582 V=800.0 PL=0
MOVL C01583 V=800.0 PL=0
MOVL C01584 V=800.0 PL=0
MOVL C01585 V=800.0 PL=0
MOVL C01586 V=800.0 PL=0
MOVL C01587 V=800.0 PL=0
MOVL C01588 V=800.0 PL=0
MOVL C01589 V=800.0 PL=0
MOVL C01590 V=800.0 PL=0
MOVL C01591 V=800.0 PL=0
MOVL C01592 V=800.0 PL=0
MOVL C01593 V=800.0 PL=0
MOVL C01594 V=800.0 PL=0
MOVL C01595 V=800.0 PL=0
MOVL C01596 V=800.0 PL=0
MOVL C01597 V=800.0 PL=0
MOVL C01598 V=800.0 PL=0
MOVL C01599 V=800.0 PL=0
MOVL C01600 V=800.0 PL=0
MOVL C01601 V=800.0 PL=0
MOVL C01602 V=800.0 PL=0
MOVL C01603 V=800.0 PL=0
MOVL C01604 V=800.0 PL=0
MOVL C01605 V=800.0 PL=0
MOVL C01606 V=800.0 PL=0
MOVL C01607 V=800.0 PL=0
MOVL C01608 V=800.0 PL=0
MOVL C01609 V=800.0 PL=0
MOVL C01610 V=800.0 PL=0
MOVL C01611 V=800.0 PL=0
MOVL C01612 V=800.0 PL=0
MOVL C01613 V=800.0 PL=0
MOVL C01614 V=800.0 PL=0
MOVL C01615 V=800.0 PL=0
MOVL C01616 V=800.0 PL=0
MOVL C01617 V=800.0 PL=0
MOVL C01618 V=800.0 PL=0
MOVL C01619 V=800.0 PL=0
MOVL C01620 V=800.0 PL=0
MOVL C01621 V=800.0 PL=0
MOVL C01622 V=800.0 PL=0
MOVL C01623 V=800.0 PL=0
MOVL C01624 V=800.0 PL=0
MOVL C01625 V=800.0 PL=0
MOVL C01626 V=800.0 PL=0
MOVL C01627 V=800.0 PL=0
MOVL C01628 V=800.0 PL=0
MOVL C01629 V=800.0 PL=0
MOVL C01630 V=800.0 PL=0
MOVL C01631 V=800.0 PL=0
MOVL C01632 V=800.0 PL=0
MOVL C01633 V=800.0 PL=0
MOVL C01634 V=800.0 PL=0
MOVL C01635 V=800.0 PL=0
MOVL C01636 V=800.0 PL=0
MOVL C01637 V=800.0 PL=0
MOVL C01638 V=800.0 PL=0
MOVL C01639 V=800.0 PL=0
MOVL C01640 V=800.0 PL=0
MOVL C01641 V=800.0 PL=0
MOVL C01642 V=800.0 PL=0
MOVL C01643 V=800.0 PL=0
MOVL C01644 V=800.0 PL=0
MOVL C01645 V=800.0 PL=0
MOVL C01646 V=800.0 PL=0
MOVL C01647 V=800.0 PL=0
MOVL C01648 V=800.0 PL=0
MOVL C01649 V=800.0 PL=0
MOVL C01650 V=800.0 PL=0
MOVL C01651 V=800.0 PL=0
MOVL C01652 V=800.0 PL=0
MOVL C01653 V=800.0 PL=0
MOVL C01654 V=800.0 PL=0
MOVL C01655 V=800.0 PL=0
MOVL C01656 V=800.0 PL=0
MOVL C01657 V=800.0 PL=0
MOVL C01658 V=800.0 PL=0
MOVL C01659 V=800.0 PL=0
MOVL C01660 V=800.0 PL=0
MOVL C01661 V=800.0 PL=0
MOVL C01662 V=800.0 PL=0
MOVL C01663 V=800.0 PL=0
MOVL C01664 V=800.0 PL=0
MOVL C01665 V=800.0 PL=0
MOVL C01666 V=800.0 PL=0
MOVL C01667 V=800.0 PL=0
MOVL C01668 V=800.0 PL=0
MOVL C01669 V=800.0 PL=0
MOVL C01670 V=800.0 PL=0
MOVL C01671 V=800.0 PL=0
MOVL C01672 V=800.0 PL=0
MOVL C01673 V=800.0 PL=0
MOVL C01674 V=800.0 PL=0
MOVL C01675 V=800.0 PL=0
MOVL C01676 V=800.0 PL=0
MOVL C01677 V=800.0 PL=0
MOVL C01678 V=800.0 PL=0
MOVL C01679 V=800.0 PL=0
MOVL C01680 V=800.0 PL=0
MOVL C01681 V=800.0 PL=0
MOVL C01682 V=800.0 PL=0
MOVL C01683 V=800.0 PL=0
MOVL C01684 V=800.0 PL=0
MOVL C01685 V=800.0 PL=0
MOVL C01686 V=800.0 PL=0
MOVL C01687 V=800.0 PL=0
MOVL C01688 V=800.0 PL=0
MOVL C01689 V=800.0 PL=0
MOVL C01690 V=800.0 PL=0
MOVL C01691 V=800.0 PL=0
MOVL C01692 V=800.0 PL=0
MOVL C01693 V=800.0 PL=0
MOVL C01694 V=800.0 PL=0
MOVL C01695 V=800.0 PL=0
MOVL C01696 V=800.0 PL=0
MOVL C01697 V=800.0 PL=0
MOVL C01698 V=800.0 PL=0
MOVL C01699 V=800.0 PL=0
MOVL C01700 V=800.0 PL=0
MOVL C01701 V=800.0 PL=0
MOVL C01702 V=800.0 PL=0
MOVL C01703 V=800.0 PL=0
MOVL C01704 V=800.0 PL=0
MOVL C01705 V=800.0 PL=0
MOVL C01706 V=800.0 PL=0
MOVL C01707 V=800.0 PL=0
MOVL C01708 V=800.0 PL=0
MOVL C01709 V=800.0 PL=0
MOVL C01710 V=800.0 PL=0
MOVL C01711 V=800.0 PL=0
MOVL C01712 V=800.0 PL=0
MOVL C01713 V=800.0 PL=0
MOVL C01714 V=800.0 PL=0
MOVL C01715 V=800.0 PL=0
MOVL C01716 V=800.0 PL=0
MOVL C01717 V=800.0 PL=0
MOVL C01718 V=800.0 PL=0
MOVL C01719 V=800.0 PL=0
MOVL C01720 V=800.0 PL=0
MOVL C01721 V=800.0 PL=0
MOVL C01722 V=800.0 PL=0
MOVL C01723 V=800.0 PL=0
MOVL C01724 V=800.0 PL=0
MOVL C01725 V=800.0 PL=0
MOVL C01726 V=800.0 PL=0
MOVL C01727 V=800.0 PL=0
MOVL C01728 V=800.0 PL=0
MOVL C01729 V=800.0 PL=0
MOVL C01730 V=800.0 PL=0
MOVL C01731 V=800.0 PL=0
MOVL C01732 V=800.0 PL=0
MOVL C01733 V=800.0 PL=0
MOVL C01734 V=800.0 PL=0
MOVL C01735 V=800.0 PL=0
MOVL C01736 V=800.0 PL=0
MOVL C01737 V=800.0 PL=0
MOVL C01738 V=800.0 PL=0
MOVL C01739 V=800.0 PL=0
MOVL C01740 V=800.0 PL=0
MOVL C01741 V=800.0 PL=0
MOVL C01742 V=800.0 PL=0
MOVL C01743 V=800.0 PL=0
MOVL C01744 V=800.0 PL=0
MOVL C01745 V=800.0 PL=0
MOVL C01746 V=800.0 PL=0
MOVL C01747 V=800.0 PL=0
MOVL C01748 V=800.0 PL=0
MOVL C01749 V=800.0 PL=0
MOVL C01750 V=800.0 PL=0
MOVL C01751 V=800.0 PL=0
MOVL C01752 V=800.0 PL=0
MOVL C01753 V=800.0 PL=0
MOVL C01754 V=800.0 PL=0
MOVL C01755 V=800.0 PL=0
MOVL C01756 V=800.0 PL=0
MOVL C01757 V=800.0 PL=0
MOVL C01758 V=800.0 PL=0
MOVL C01759 V=800.0 PL=0
MOVL C01760 V=800.0 PL=0
MOVL C01761 V=800.0 PL=0
MOVL C01762 V=800.0 PL=0
MOVL C01763 V=800.0 PL=0
MOVL C01764 V=800.0 PL=0
MOVL C01765 V=800.0 PL=0
MOVL C01766 V=800.0 PL=0
MOVL C01767 V=800.0 PL=0
MOVL C01768 V=800.0 PL=0
MOVL C01769 V=800.0 PL=0
MOVL C01770 V=800.0 PL=0
MOVL C01771 V=800.0 PL=0
MOVL C01772 V=800.0 PL=0
MOVL C01773 V=800.0 PL=0
MOVL C01774 V=800.0 PL=0
MOVL C01775 V=800.0 PL=0
MOVL C01776 V=800.0 PL=0
MOVL C01777 V=800.0 PL=0
MOVL C01778 V=800.0 PL=0
MOVL C01779 V=800.0 PL=0
MOVL C01780 V=800.0 PL=0
MOVL C01781 V=800.0 PL=0
MOVL C01782 V=800.0 PL=0
MOVL C01783 V=800.0 PL=0
MOVL C01784 V=800.0 PL=0
MOVL C01785 V=800.0 PL=0
MOVL C01786 V=800.0 PL=0
MOVL C01787 V=800.0 PL=0
MOVL C01788 V=800.0 PL=0
MOVL C01789 V=800.0 PL=0
MOVL C01790 V=800.0 PL=0
MOVL C01791 V=800.0 PL=0
MOVL C01792 V=800.0 PL=0
MOVL C01793 V=800.0 PL=0
MOVL C01794 V=800.0 PL=0
MOVL C01795 V=800.0 PL=0
MOVL C01796 V=800.0 PL=0
MOVL C01797 V=800.0 PL=0
MOVL C01798 V=800.0 PL=0
MOVL C01799 V=800.0 PL=0
MOVL C01800 V=800.0 PL=0
MOVL C01801 V=800.0 PL=0
MOVL C01802 V=800.0 PL=0
MOVL C01803 V=800.0 PL=0
MOVL C01804 V=800.0 PL=0
MOVL C01805 V=800.0 PL=0
MOVL C01806 V=800.0 PL=0
MOVL C01807 V=800.0 PL=0
MOVL C01808 V=800.0 PL=0
MOVL C01809 V=800.0 PL=0
MOVL C01810 V=800.0 PL=0
MOVL C01811 V=800.0 PL=0
MOVL C01812 V=800.0 PL=0
MOVL C01813 V=800.0 PL=0
MOVL C01814 V=800.0 PL=0
MOVL C01815 V=800.0 PL=0
MOVL C01816 V=800.0 PL=0
MOVL C01817 V=800.0 PL=0
MOVL C01818 V=800.0 PL=0
MOVL C01819 V=800.0 PL=0
MOVL C01820 V=800.0 PL=0
MOVL C01821 V=800.0 PL=0
MOVL C01822 V=800.0 PL=0
MOVL C01823 V=800.0 PL=0
MOVL C01824 V=800.0 PL=0
MOVL C01825 V=800.0 PL=0
MOVL C01826 V=800.0 PL=0
MOVL C01827 V=800.0 PL=0
MOVL C01828 V=800.0 PL=0
MOVL C01829 V=800.0 PL=0
MOVL C01830 V=800.0 PL=0
MOVL C01831 V=800.0 PL=0
MOVL C01832 V=800.0 PL=0
MOVL C01833 V=800.0 PL=0
MOVL C01834 V=800.0 PL=0
MOVL C01835 V=800.0 PL=0
MOVL C01836 V=800.0 PL=0
MOVL C01837 V=800.0 PL=0
MOVL C01838 V=800.0 PL=0
MOVL C01839 V=800.0 PL=0
MOVL C01840 V=800.0 PL=0
MOVL C01841 V=800.0 PL=0
MOVL C01842 V=800.0 PL=0
MOVL C01843 V=800.0 PL=0
MOVL C01844 V=800.0 PL=0
MOVL C01845 V=800.0 PL=0
MOVL C01846 V=800.0 PL=0
MOVL C01847 V=800.0 PL=0
MOVL C01848 V=800.0 PL=0
MOVL C01849 V=800.0 PL=0
MOVL C01850 V=800.0 PL=0
MOVL C01851 V=800.0 PL=0
MOVL C01852 V=800.0 PL=0
MOVL C01853 V=800.0 PL=0
MOVL C01854 V=800.0 PL=0
MOVL C01855 V=800.0 PL=0
MOVL C01856 V=800.0 PL=0
MOVL C01857 V=800.0 PL=0
MOVL C01858 V=800.0 PL=0
MOVL C01859 V=800.0 PL=0
MOVL C01860 V=800.0 PL=0
MOVL C01861 V=800.0 PL=0
MOVL C01862 V=800.0 PL=0
MOVL C01863 V=800.0 PL=0
MOVL C01864 V=800.0 PL=0
MOVL C01865 V=800.0 PL=0
MOVL C01866 V=800.0 PL=0
MOVL C01867 V=800.0 PL=0
MOVL C01868 V=800.0 PL=0
MOVL C01869 V=800.0 PL=0
MOVL C01870 V=800.0 PL=0
MOVL C01871 V=800.0 PL=0
MOVL C01872 V=800.0 PL=0
MOVL C01873 V=800.0 PL=0
MOVL C01874 V=800.0 PL=0
MOVL C01875 V=800.0 PL=0
MOVL C01876 V=800.0 PL=0
MOVL C01877 V=800.0 PL=0
MOVL C01878 V=800.0 PL=0
MOVL C01879 V=800.0 PL=0
MOVL C01880 V=800.0 PL=0
MOVL C01881 V=800.0 PL=0
MOVL C01882 V=800.0 PL=0
MOVL C01883 V=800.0 PL=0
MOVL C01884 V=800.0 PL=0
MOVL C01885 V=800.0 PL=0
MOVL C01886 V=800.0 PL=0
MOVL C01887 V=800.0 PL=0
MOVL C01888 V=800.0 PL=0
MOVL C01889 V=800.0 PL=0
MOVL C01890 V=800.0 PL=0
MOVL C01891 V=800.0 PL=0
MOVL C01892 V=800.0 PL=0
MOVL C01893 V=800.0 PL=0
MOVL C01894 V=800.0 PL=0
MOVL C01895 V=800.0 PL=0
MOVL C01896 V=800.0 PL=0
MOVL C01897 V=800.0 PL=0
MOVL C01898 V=800.0 PL=0
MOVL C01899 V=800.0 PL=0
MOVL C01900 V=800.0 PL=0
MOVL C01901 V=800.0 PL=0
MOVL C01902 V=800.0 PL=0
MOVL C01903 V=800.0 PL=0
MOVL C01904 V=800.0 PL=0
MOVL C01905 V=800.0 PL=0
MOVL C01906 V=800.0 PL=0
MOVL C01907 V=800.0 PL=0
MOVL C01908 V=800.0 PL=0
MOVL C01909 V=800.0 PL=0
MOVL C01910 V=800.0 PL=0
MOVL C01911 V=800.0 PL=0
MOVL C01912 V=800.0 PL=0
MOVL C01913 V=800.0 PL=0
MOVL C01914 V=800.0 PL=0
MOVL C01915 V=800.0 PL=0
MOVL C01916 V=800.0 PL=0
MOVL C01917 V=800.0 PL=0
MOVL C01918 V=800.0 PL=0
MOVL C01919 V=800.0 PL=0
MOVL C01920 V=800.0 PL=0
MOVL C01921 V=800.0 PL=0
MOVL C01922 V=800.0 PL=0
MOVL C01923 V=800.0 PL=0
MOVL C01924 V=800.0 PL=0
MOVL C01925 V=800.0 PL=0
MOVL C01926 V=800.0 PL=0
MOVL C01927 V=800.0 PL=0
MOVL C01928 V=800.0 PL=0
MOVL C01929 V=800.0 PL=0
MOVL C01930 V=800.0 PL=0
MOVL C01931 V=800.0 PL=0
MOVL C01932 V=800.0 PL=0
MOVL C01933 V=800.0 PL=0
MOVL C01934 V=800.0 PL=0
MOVL C01935 V=800.0 PL=0
MOVL C01936 V=800.0 PL=0
MOVL C01937 V=800.0 PL=0
MOVL C01938 V=800.0 PL=0
MOVL C01939 V=800.0 PL=0
MOVL C01940 V=800.0 PL=0
MOVL C01941 V=800.0 PL=0
MOVL C01942 V=800.0 PL=0
MOVL C01943 V=800.0 PL=0
MOVL C01944 V=800.0 PL=0
MOVL C01945 V=800.0 PL=0
MOVL C01946 V=800.0 PL=0
MOVL C01947 V=800.0 PL=0
MOVL C01948 V=800.0 PL=0
MOVL C01949 V=800.0 PL=0
MOVL C01950 V=800.0 PL=0
MOVL C01951 V=800.0 PL=0
MOVL C01952 V=800.0 PL=0
MOVL C01953 V=800.0 PL=0
MOVL C01954 V=800.0 PL=0
MOVL C01955 V=800.0 PL=0
MOVL C01956 V=800.0 PL=0
MOVL C01957 V=800.0 PL=0
MOVL C01958 V=800.0 PL=0
MOVL C01959 V=800.0 PL=0
MOVL C01960 V=800.0 PL=0
MOVL C01961 V=800.0 PL=0
MOVL C01962 V=800.0 PL=0
MOVL C01963 V=800.0 PL=0
MOVL C01964 V=800.0 PL=0
MOVL C01965 V=800.0 PL=0
MOVL C01966 V=800.0 PL=0
MOVL C01967 V=800.0 PL=0
MOVL C01968 V=800.0 PL=0
MOVL C01969 V=800.0 PL=0
MOVL C01970 V=800.0 PL=0
MOVL C01971 V=800.0 PL=0
MOVL C01972 V=800.0 PL=0
MOVL C01973 V=800.0 PL=0
MOVL C01974 V=800.0 PL=0
MOVL C01975 V=800.0 PL=0
MOVL C01976 V=800.0 PL=0
MOVL C01977 V=800.0 PL=0
MOVL C01978 V=800.0 PL=0
MOVL C01979 V=800.0 PL=0
MOVL C01980 V=800.0 PL=0
MOVL C01981 V=800.0 PL=0
MOVL C01982 V=800.0 PL=0
MOVL C01983 V=800.0 PL=0
MOVL C01984 V=800.0 PL=0
MOVL C01985 V=800.0 PL=0
MOVL C01986 V=800.0 PL=0
MOVL C01987 V=800.0 PL=0
MOVL C01988 V=800.0 PL=0
MOVL C01989 V=800.0 PL=0
MOVL C01990 V=800.0 PL=0
MOVL C01991 V=800.0 PL=0
MOVL C01992 V=800.0 PL=0
MOVL C01993 V=800.0 PL=0
MOVL C01994 V=800.0 PL=0
MOVL C01995 V=800.0 PL=0
MOVL C01996 V=800.0 PL=0
MOVL C01997 V=800.0 PL=0
MOVL C01998 V=800.0 PL=0
MOVL C01999 V=800.0 PL=0
MOVL C02000 V=800.0 PL=0
MOVL C02001 V=800.0 PL=0
MOVL C02002 V=800.0 PL=0
MOVL C02003 V=800.0 PL=0
MOVL C02004 V=800.0 PL=0
MOVL C02005 V=800.0 PL=0
MOVL C02006 V=800.0 PL=0
MOVL C02007 V=800.0 PL=0
MOVL C02008 V=800.0 PL=0
MOVL C02009 V=800.0 PL=0
MOVL C02010 V=800.0 PL=0
MOVL C02011 V=800.0 PL=0
MOVL C02012 V=800.0 PL=0
MOVL C02013 V=800.0 PL=0
MOVL C02014 V=800.0 PL=0
MOVL C02015 V=800.0 PL=0
MOVL C02016 V=800.0 PL=0
MOVL C02017 V=800.0 PL=0
MOVL C02018 V=800.0 PL=0
MOVL C02019 V=800.0 PL=0
MOVL C02020 V=800.0 PL=0
MOVL C02021 V=800.0 PL=0
MOVL C02022 V=800.0 PL=0
MOVL C02023 V=800.0 PL=0
MOVL C02024 V=800.0 PL=0
MOVL C02025 V=800.0 PL=0
MOVL C02026 V=800.0 PL=0
MOVL C02027 V=800.0 PL=0
MOVL C02028 V=800.0 PL=0
MOVL C02029 V=800.0 PL=0
MOVL C02030 V=800.0 PL=0
MOVL C02031 V=800.0 PL=0
MOVL C02032 V=800.0 PL=0
MOVL C02033 V=800.0 PL=0
MOVL C02034 V=800.0 PL=0
MOVL C02035 V=800.0 PL=0
MOVL C02036 V=800.0 PL=0
MOVL C02037 V=800.0 PL=0
MOVL C02038 V=800.0 PL=0
MOVL C02039 V=800.0 PL=0
MOVL C02040 V=800.0 PL=0
MOVL C02041 V=800.0 PL=0
MOVL C02042 V=800.0 PL=0
MOVL C02043 V=800.0 PL=0
MOVL C02044 V=800.0 PL=0
MOVL C02045 V=800.0 PL=0
MOVL C02046 V=800.0 PL=0
MOVL C02047 V=800.0 PL=0
MOVL C02048 V=800.0 PL=0
MOVL C02049 V=800.0 PL=0
MOVL C02050 V=800.0 PL=0
MOVL C02051 V=800.0 PL=0
MOVL C02052 V=800.0 PL=0
MOVL C02053 V=800.0 PL=0
MOVL C02054 V=800.0 PL=0
MOVL C02055 V=800.0 PL=0
MOVL C02056 V=800.0 PL=0
MOVL C02057 V=800.0 PL=0
MOVL C02058 V=800.0 PL=0
MOVL C02059 V=800.0 PL=0
MOVL C02060 V=800.0 PL=0
MOVL C02061 V=800.0 PL=0
MOVL C02062 V=800.0 PL=0
MOVL C02063 V=800.0 PL=0
MOVL C02064 V=800.0 PL=0
MOVL C02065 V=800.0 PL=0
MOVL C02066 V=800.0 PL=0
MOVL C02067 V=800.0 PL=0
MOVL C02068 V=800.0 PL=0
MOVL C02069 V=800.0 PL=0
MOVL C02070 V=800.0 PL=0
MOVL C02071 V=800.0 PL=0
MOVL C02072 V=800.0 PL=0
MOVL C02073 V=800.0 PL=0
MOVL C02074 V=800.0 PL=0
MOVL C02075 V=800.0 PL=0
MOVL C02076 V=800.0 PL=0
MOVL C02077 V=800.0 PL=0
MOVL C02078 V=800.0 PL=0
MOVL C02079 V=800.0 PL=0
MOVL C02080 V=800.0 PL=0
MOVL C02081 V=800.0 PL=0
MOVL C02082 V=800.0 PL=0
MOVL C02083 V=800.0 PL=0
MOVL C02084 V=800.0 PL=0
MOVL C02085 V=800.0 PL=0
MOVL C02086 V=800.0 PL=0
MOVL C02087 V=800.0 PL=0
MOVL C02088 V=800.0 PL=0
MOVL C02089 V=800.0 PL=0
MOVL C02090 V=800.0 PL=0
MOVL C02091 V=800.0 PL=0
MOVL C02092 V=800.0 PL=0
MOVL C02093 V=800.0 PL=0
MOVL C02094 V=800.0 PL=0
MOVL C02095 V=800.0 PL=0
MOVL C02096 V=800.0 PL=0
MOVL C02097 V=800.0 PL=0
MOVL C02098 V=800.0 PL=0
MOVL C02099 V=800.0 PL=0
MOVL C02100 V=800.0 PL=0
MOVL C02101 V=800.0 PL=0
MOVL C02102 V=800.0 PL=0
MOVL C02103 V=800.0 PL=0
MOVL C02104 V=800.0 PL=0
MOVL C02105 V=800.0 PL=0
MOVL C02106 V=800.0 PL=0
MOVL C02107 V=800.0 PL=0
MOVL C02108 V=800.0 PL=0
MOVL C02109 V=800.0 PL=0
MOVL C02110 V=800.0 PL=0
MOVL C02111 V=800.0 PL=0
